C09107=1078.926,391.055,397.098,176.330,30.069,155.273
C09108=1078.920,390.808,397.137,176.326,30.062,155.271
C09109=1078.913,390.562,397.177,176.323,30.054,155.269
C09110=1078.906,390.315,397.216,176.319,30.047,155.268
C09111=1078.900,390.068,397.255,176.314,30.039,155.266
C09112=1078.893,389.821,397.295,176.311,30.032,155.265
C09113=1078.886,389.575,397.333,176.307,30.024,155.263
C09114=1078.880,389.327,397.373,176.303,30.016,155.262
C09115=1078.873,389.081,397.412,176.299,30.009,155.260
C09116=1078.866,388.834,397.451,176.295,30.002,155.259
C09117=1078.860,388.587,397.491,176.291,29.994,155.257
C09118=1078.853,388.340,397.529,176.287,29.986,155.256
C09119=1078.846,388.094,397.569,176.284,29.979,155.254
C09120=1078.840,387.847,397.608,176.279,29.972,155.253
C09121=1078.833,387.600,397.647,176.275,29.964,155.251
C09122=1078.827,387.354,397.686,176.271,29.957,155.250
C09123=1078.821,387.107,397.725,176.268,29.949,155.248
C09124=1078.814,386.860,397.764,176.264,29.942,155.247
C09125=1078.807,386.613,397.803,176.259,29.934,155.245
C09126=1078.801,386.366,397.842,176.256,29.928,155.244
C09127=1078.794,386.119,397.881,176.252,29.920,155.242
C09128=1078.788,385.886,397.918,176.249,29.913,155.241
C09129=1078.782,385.653,397.955,176.245,29.906,155.240
C09130=1078.776,385.419,397.991,176.241,29.899,155.238
C09131=1078.769,385.185,398.029,176.238,29.892,155.237
C09132=1078.764,384.951,398.065,176.234,29.886,155.236
C09133=1078.758,384.718,398.102,176.231,29.879,155.234
C09134=1078.752,384.484,398.139,176.226,29.872,155.233
C09135=1078.746,384.251,398.175,176.223,29.865,155.232
C09136=1078.739,384.004,398.214,176.219,29.858,155.230
C09137=1078.732,383.757,398.252,176.216,29.851,155.229
C09138=1078.726,383.509,398.292,176.211,29.844,155.227
C09139=1078.720,383.263,398.330,176.208,29.837,155.226
C09140=1078.713,383.017,398.369,176.204,29.829,155.224
C09141=1078.707,382.769,398.407,176.200,29.822,155.223
C09142=1078.701,382.523,398.446,176.197,29.815,155.222
C09143=1078.694,382.276,398.485,176.192,29.808,155.220
C09144=1078.688,382.028,398.523,176.189,29.801,155.219
C09145=1078.681,381.782,398.562,176.185,29.794,155.217
C09146=1078.675,381.535,398.601,176.182,29.787,155.216
C09147=1078.668,381.288,398.639,176.178,29.780,155.215
C09148=1078.662,381.041,398.678,176.173,29.773,155.213
C09149=1078.655,380.795,398.715,176.170,29.766,155.212
C09150=1078.648,380.548,398.754,176.166,29.759,155.211
C09151=1078.642,380.300,398.792,176.163,29.752,155.209
C09152=1078.635,380.054,398.830,176.158,29.745,155.208
C09153=1078.629,379.807,398.868,176.155,29.739,155.207
C09154=1078.622,379.559,398.906,176.151,29.731,155.205
C09155=1078.616,379.313,398.945,176.148,29.725,155.204
C09156=1078.610,379.066,398.983,176.144,29.718,155.203
C09157=1078.604,378.819,399.021,176.140,29.711,155.201
C09158=1078.597,378.572,399.060,176.136,29.704,155.200
C09159=1078.591,378.325,399.098,176.133,29.697,155.198
C09160=1078.584,378.078,399.135,176.129,29.691,155.197
C09161=1078.577,377.832,399.174,176.125,29.684,155.196
C09162=1078.571,377.585,399.211,176.121,29.677,155.194
C09163=1078.565,377.337,399.250,176.118,29.670,155.193
C09164=1078.559,377.091,399.287,176.114,29.664,155.192
C09165=1078.552,376.843,399.325,176.111,29.657,155.191
C09166=1078.546,376.596,399.363,176.106,29.650,155.189
C09167=1078.539,376.350,399.401,176.103,29.643,155.188
C09168=1078.533,376.103,399.439,176.099,29.637,155.187
C09169=1078.526,375.856,399.477,176.096,29.630,155.185
C09170=1078.520,375.609,399.515,176.092,29.623,155.184
C09171=1078.514,375.362,399.553,176.088,29.617,155.183
C09172=1078.507,375.115,399.590,176.084,29.610,155.182
C09173=1078.501,374.868,399.628,176.081,29.604,155.180
C09174=1078.495,374.621,399.666,176.077,29.597,155.179
C09175=1078.489,374.374,399.704,176.074,29.590,155.178
C09176=1078.482,374.127,399.742,176.069,29.584,155.176
C09177=1078.476,373.880,399.779,176.066,29.577,155.175
C09178=1078.469,373.633,399.817,176.063,29.571,155.174
C09179=1078.464,373.386,399.854,176.059,29.564,155.173
C09180=1078.456,373.138,399.892,176.055,29.558,155.171
C09181=1078.451,372.892,399.930,176.051,29.551,155.170
C09182=1078.443,372.645,399.967,176.048,29.545,155.169
C09183=1078.437,372.398,400.005,176.044,29.538,155.168
C09184=1078.432,372.178,400.038,176.041,29.533,155.167
C09185=1078.427,371.959,400.071,176.038,29.528,155.166
C09186=1078.420,371.740,400.104,176.035,29.522,155.164
C09187=1078.415,371.520,400.137,176.032,29.516,155.163
C09188=1078.409,371.301,400.171,176.028,29.510,155.162
C09189=1078.404,371.082,400.204,176.025,29.504,155.161
C09190=1078.398,370.862,400.238,176.022,29.499,155.160
C09191=1078.392,370.643,400.269,176.018,29.493,155.159
C09192=1078.386,370.396,400.308,176.015,29.487,155.158
C09193=1078.379,370.149,400.345,176.011,29.481,155.157
C09194=1078.374,369.902,400.382,176.008,29.475,155.156
C09195=1078.366,369.655,400.419,176.004,29.468,155.154
C09196=1078.361,369.407,400.456,176.000,29.462,155.153
C09197=1078.354,369.161,400.493,175.997,29.456,155.152
C09198=1078.348,368.913,400.531,175.993,29.449,155.151
C09199=1078.341,368.666,400.568,175.990,29.443,155.149
C09200=1078.336,368.419,400.605,175.986,29.437,155.148
C09201=1078.329,368.172,400.642,175.982,29.431,155.147
C09202=1078.322,367.925,400.679,175.979,29.424,155.146
C09203=1078.316,367.677,400.716,175.976,29.418,155.145
C09204=1078.310,367.431,400.753,175.972,29.412,155.144
C09205=1078.304,367.184,400.790,175.968,29.406,155.142
C09206=1078.298,366.937,400.827,175.965,29.400,155.141
C09207=1078.292,366.688,400.864,175.961,29.393,155.140
C09208=1078.285,366.442,400.901,175.958,29.387,155.139
C09209=1078.279,366.195,400.938,175.954,29.381,155.138
C09210=1078.273,365.948,400.975,175.950,29.375,155.137
C09211=1078.267,365.701,401.011,175.947,29.369,155.135
C09212=1078.261,365.454,401.049,175.944,29.363,155.134
C09213=1078.254,365.206,401.086,175.940,29.357,155.133
C09214=1078.248,364.959,401.122,175.936,29.351,155.132
C09215=1078.241,364.712,401.159,175.933,29.344,155.131
C09216=1078.236,364.465,401.196,175.930,29.338,155.130
C09217=1078.229,364.218,401.232,175.926,29.333,155.129
C09218=1078.223,363.970,401.269,175.922,29.327,155.128
C09219=1078.216,363.723,401.305,175.919,29.321,155.126
C09220=1078.210,363.476,401.342,175.915,29.314,155.125
C09221=1078.204,363.228,401.379,175.912,29.309,155.124
C09222=1078.198,362.981,401.415,175.908,29.303,155.123
C09223=1078.191,362.734,401.452,175.904,29.296,155.122
C09224=1078.185,362.487,401.488,175.901,29.291,155.121
C09225=1078.179,362.240,401.525,175.898,29.285,155.120
C09226=1078.172,361.993,401.561,175.895,29.279,155.119
C09227=1078.165,361.745,401.598,175.890,29.273,155.118
C09228=1078.160,361.498,401.635,175.887,29.267,155.116
C09229=1078.154,361.250,401.671,175.884,29.261,155.115
C09230=1078.148,361.003,401.707,175.881,29.256,155.114
C09231=1078.141,360.756,401.744,175.876,29.249,155.113
C09232=1078.135,360.509,401.780,175.873,29.244,155.112
C09233=1078.128,360.262,401.817,175.870,29.238,155.111
C09234=1078.122,360.014,401.852,175.867,29.232,155.110
C09235=1078.116,359.767,401.889,175.862,29.226,155.109
C09236=1078.110,359.520,401.925,175.859,29.220,155.108
C09237=1078.104,359.273,401.961,175.856,29.215,155.107
C09238=1078.097,359.026,401.997,175.853,29.209,155.106
C09239=1078.091,358.778,402.034,175.849,29.203,155.105
C09240=1078.086,358.567,402.064,175.846,29.198,155.104
C09241=1078.080,358.356,402.095,175.843,29.193,155.103
C09242=1078.075,358.145,402.126,175.840,29.189,155.102
C09243=1078.070,357.934,402.156,175.837,29.184,155.101
C09244=1078.064,357.722,402.187,175.834,29.178,155.100
C09245=1078.059,357.511,402.218,175.831,29.174,155.099
C09246=1078.053,357.300,402.249,175.828,29.169,155.098
C09247=1078.048,357.089,402.280,175.826,29.164,155.097
C09248=1078.042,356.842,402.315,175.822,29.158,155.096
C09249=1078.036,356.595,402.352,175.818,29.153,155.095
C09250=1078.030,356.347,402.387,175.815,29.147,155.094
C09251=1078.024,356.100,402.424,175.812,29.142,155.093
C09252=1078.018,355.852,402.460,175.809,29.136,155.092
C09253=1078.012,355.604,402.495,175.805,29.131,155.091
C09254=1078.005,355.357,402.532,175.801,29.125,155.090
C09255=1077.998,355.110,402.567,175.798,29.119,155.089
C09256=1077.993,354.863,402.602,175.795,29.114,155.088
C09257=1077.987,354.616,402.639,175.791,29.108,155.087
C09258=1077.981,354.368,402.674,175.788,29.102,155.086
C09259=1077.975,354.121,402.710,175.785,29.097,155.085
C09260=1077.968,353.874,402.747,175.781,29.091,155.084
C09261=1077.962,353.626,402.782,175.777,29.085,155.083
C09262=1077.956,353.379,402.817,175.774,29.080,155.082
C09263=1077.950,353.132,402.853,175.771,29.074,155.081
C09264=1077.944,352.884,402.889,175.768,29.069,155.080
C09265=1077.937,352.637,402.924,175.764,29.063,155.079
C09266=1077.931,352.389,402.960,175.760,29.058,155.078
C09267=1077.925,352.142,402.996,175.757,29.052,155.077
C09268=1077.918,351.894,403.031,175.754,29.047,155.076
C09269=1077.913,351.647,403.066,175.750,29.041,155.075
C09270=1077.907,351.400,403.102,175.747,29.036,155.074
C09271=1077.900,351.152,403.137,175.744,29.031,155.073
C09272=1077.894,350.905,403.173,175.741,29.025,155.072
C09273=1077.888,350.657,403.209,175.737,29.020,155.071
C09274=1077.882,350.410,403.243,175.733,29.014,155.070
C09275=1077.876,350.163,403.279,175.730,29.009,155.069
C09276=1077.869,349.915,403.314,175.727,29.003,155.068
C09277=1077.863,349.668,403.350,175.724,28.998,155.067
C09278=1077.857,349.420,403.384,175.720,28.993,155.066
C09279=1077.851,349.173,403.420,175.717,28.987,155.065
C09280=1077.845,348.925,403.456,175.714,28.982,155.064
C09281=1077.839,348.678,403.490,175.710,28.977,155.064
C09282=1077.833,348.431,403.526,175.707,28.971,155.062
C09283=1077.826,348.183,403.561,175.704,28.966,155.062
C09284=1077.820,347.935,403.596,175.700,28.960,155.061
C09285=1077.814,347.688,403.631,175.697,28.955,155.060
C09286=1077.808,347.441,403.667,175.693,28.950,155.059
C09287=1077.801,347.193,403.702,175.690,28.944,155.058
C09288=1077.796,346.946,403.737,175.687,28.939,155.057
C09289=1077.789,346.698,403.772,175.684,28.934,155.056
C09290=1077.783,346.451,403.807,175.680,28.929,155.055
C09291=1077.778,346.203,403.841,175.677,28.923,155.054
C09292=1077.772,345.956,403.877,175.674,28.918,155.053
C09293=1077.765,345.709,403.912,175.671,28.913,155.052
C09294=1077.759,345.461,403.946,175.667,28.908,155.051
C09295=1077.753,345.213,403.982,175.664,28.903,155.050
C09296=1077.748,345.004,404.011,175.661,28.898,155.050
C09297=1077.743,344.794,404.041,175.658,28.894,155.049
C09298=1077.738,344.585,404.071,175.656,28.889,155.048
C09299=1077.733,344.375,404.100,175.653,28.885,155.047
C09300=1077.727,344.166,404.129,175.650,28.880,155.046
C09301=1077.722,343.956,404.159,175.647,28.876,155.046
C09302=1077.717,343.747,404.188,175.645,28.871,155.045
C09303=1077.712,343.537,404.217,175.641,28.867,155.044
C09304=1077.705,343.290,404.253,175.638,28.862,155.043
C09305=1077.699,343.042,404.287,175.635,28.857,155.042
C09306=1077.693,342.795,404.322,175.631,28.852,155.041
C09307=1077.687,342.547,404.357,175.628,28.847,155.040
C09308=1077.681,342.299,404.391,175.625,28.842,155.040
C09309=1077.674,342.052,404.426,175.622,28.836,155.039
C09310=1077.669,341.804,404.461,175.618,28.831,155.038
C09311=1077.663,341.556,404.495,175.615,28.826,155.037
C09312=1077.656,341.310,404.530,175.612,28.821,155.036
C09313=1077.650,341.062,404.564,175.609,28.816,155.035
C09314=1077.644,340.815,404.598,175.605,28.811,155.034
C09315=1077.638,340.566,404.633,175.602,28.806,155.033
C09316=1077.632,340.320,404.668,175.599,28.801,155.032
C09317=1077.626,340.072,404.702,175.596,28.795,155.031
C09318=1077.620,339.824,404.736,175.592,28.790,155.031
C09319=1077.613,339.576,404.771,175.589,28.786,155.030
C09320=1077.608,339.329,404.806,175.586,28.781,155.029
C09321=1077.602,339.081,404.840,175.582,28.775,155.028
C09322=1077.596,338.833,404.874,175.580,28.771,155.027
C09323=1077.590,338.587,404.909,175.577,28.765,155.026
C09324=1077.583,338.339,404.943,175.574,28.760,155.025
C09325=1077.577,338.092,404.977,175.570,28.756,155.025
C09326=1077.571,337.844,405.012,175.567,28.751,155.024
C09327=1077.565,337.596,405.046,175.564,28.745,155.023
C09328=1077.559,337.348,405.080,175.561,28.741,155.022
C09329=1077.553,337.101,405.114,175.557,28.736,155.021
C09330=1077.547,336.854,405.148,175.554,28.730,155.020
C09331=1077.540,336.606,405.183,175.551,28.726,155.019
C09332=1077.535,336.358,405.216,175.548,28.721,155.018
C09333=1077.528,336.110,405.250,175.544,28.716,155.018
C09334=1077.523,335.863,405.284,175.541,28.711,155.017
C09335=1077.517,335.615,405.319,175.538,28.706,155.016
C09336=1077.510,335.367,405.353,175.535,28.701,155.015
C09337=1077.504,335.120,405.387,175.531,28.696,155.014
C09338=1077.499,334.873,405.421,175.528,28.691,155.013
C09339=1077.492,334.624,405.455,175.525,28.686,155.013
C09340=1077.487,334.377,405.489,175.522,28.682,155.012
C09341=1077.481,334.130,405.523,175.519,28.677,155.011
C09342=1077.474,333.882,405.557,175.516,28.672,155.010
C09343=1077.469,333.634,405.591,175.513,28.667,155.009
C09344=1077.462,333.387,405.624,175.509,28.662,155.008
C09345=1077.456,333.139,405.658,175.506,28.657,155.008
C09346=1077.450,332.891,405.693,175.503,28.652,155.007
C09347=1077.444,332.644,405.726,175.500,28.647,155.006
C09348=1077.438,332.396,405.760,175.496,28.643,155.005
C09349=1077.432,332.148,405.794,175.493,28.637,155.004
C09350=1077.426,331.900,405.828,175.491,28.633,155.003
C09351=1077.420,331.653,405.862,175.488,28.628,155.002
C09352=1077.415,331.441,405.890,175.484,28.624,155.002
C09353=1077.409,331.228,405.919,175.482,28.620,155.001
C09354=1077.404,331.017,405.947,175.479,28.616,155.000
C09355=1077.400,330.804,405.977,175.476,28.612,155.000
C09356=1077.394,330.592,406.005,175.474,28.608,154.999
C09357=1077.388,330.379,406.034,175.471,28.604,154.998
C09358=1077.383,330.167,406.063,175.468,28.599,154.998
C09359=1077.378,329.955,406.091,175.465,28.596,154.997
C09360=1077.372,329.707,406.125,175.462,28.591,154.996
C09361=1077.365,329.460,406.158,175.459,28.586,154.996
C09362=1077.360,329.212,406.192,175.457,28.582,154.995
C09363=1077.353,328.965,406.225,175.453,28.577,154.994
C09364=1077.347,328.716,406.259,175.450,28.573,154.993
C09365=1077.341,328.468,406.292,175.447,28.567,154.992
C09366=1077.335,328.221,406.326,175.443,28.563,154.992
C09367=1077.329,327.974,406.359,175.440,28.558,154.991
C09368=1077.322,327.725,406.392,175.437,28.553,154.990
C09369=1077.316,327.478,406.426,175.435,28.549,154.989
C09370=1077.310,327.230,406.459,175.431,28.544,154.988
C09371=1077.304,326.982,406.492,175.428,28.540,154.988
C09372=1077.298,326.735,406.525,175.425,28.535,154.987
C09373=1077.292,326.488,406.559,175.421,28.530,154.986
C09374=1077.285,326.239,406.592,175.418,28.526,154.985
C09375=1077.280,325.991,406.625,175.416,28.521,154.985
C09376=1077.274,325.744,406.658,175.413,28.517,154.984
C09377=1077.268,325.496,406.692,175.409,28.512,154.983
C09378=1077.261,325.249,406.725,175.406,28.507,154.982
C09379=1077.256,325.001,406.758,175.403,28.503,154.981
C09380=1077.250,324.753,406.791,175.400,28.498,154.981
C09381=1077.243,324.506,406.824,175.397,28.494,154.980
C09382=1077.237,324.257,406.858,175.394,28.489,154.979
C09383=1077.231,324.010,406.890,175.391,28.484,154.978
C09384=1077.225,323.762,406.924,175.387,28.480,154.978
C09385=1077.219,323.514,406.956,175.385,28.475,154.977
C09386=1077.213,323.266,406.990,175.382,28.471,154.976
C09387=1077.207,323.019,407.022,175.379,28.466,154.975
C09388=1077.202,322.771,407.056,175.375,28.461,154.974
C09389=1077.195,322.523,407.089,175.372,28.457,154.974
C09390=1077.189,322.276,407.121,175.370,28.452,154.973
C09391=1077.183,322.028,407.155,175.366,28.447,154.972
C09392=1077.177,321.780,407.187,175.363,28.443,154.971
C09393=1077.172,321.532,407.221,175.360,28.439,154.971
C09394=1077.165,321.285,407.253,175.358,28.434,154.970
C09395=1077.159,321.037,407.286,175.354,28.429,154.969
C09396=1077.154,320.788,407.319,175.351,28.425,154.968
C09397=1077.147,320.541,407.352,175.348,28.420,154.968
C09398=1077.141,320.293,407.384,175.345,28.416,154.967
C09399=1077.136,320.046,407.417,175.342,28.411,154.966
C09400=1077.130,319.798,407.450,175.339,28.406,154.965
C09401=1077.125,319.550,407.483,175.336,28.402,154.965
C09402=1077.118,319.302,407.515,175.333,28.398,154.964
C09403=1077.112,319.055,407.548,175.330,28.393,154.963
C09404=1077.107,318.807,407.581,175.327,28.388,154.962
C09405=1077.101,318.559,407.613,175.324,28.384,154.962
C09406=1077.094,318.311,407.646,175.321,28.379,154.961
C09407=1077.089,318.063,407.680,175.318,28.375,154.960
C09408=1077.084,317.848,407.707,175.316,28.371,154.959
C09409=1077.079,317.633,407.736,175.312,28.367,154.959
C09410=1077.073,317.417,407.764,175.310,28.363,154.958
C09411=1077.068,317.201,407.792,175.307,28.359,154.957
C09412=1077.063,316.986,407.821,175.305,28.355,154.957
C09413=1077.058,316.771,407.849,175.303,28.351,154.956
C09414=1077.054,316.555,407.877,175.299,28.347,154.956
C09415=1077.048,316.340,407.906,175.297,28.343,154.955
C09416=1077.042,316.091,407.938,175.294,28.339,154.954
C09417=1077.037,315.845,407.970,175.291,28.335,154.953
C09418=1077.030,315.597,408.003,175.288,28.330,154.953
C09419=1077.025,315.348,408.036,175.285,28.325,154.952
C09420=1077.019,315.101,408.069,175.283,28.321,154.951
C09421=1077.013,314.853,408.100,175.279,28.317,154.950
C09422=1077.008,314.605,408.133,175.276,28.312,154.950
C09423=1077.001,314.357,408.165,175.273,28.308,154.949
C09424=1076.995,314.109,408.197,175.270,28.303,154.948
C09425=1076.989,313.862,408.230,175.267,28.299,154.948
C09426=1076.983,313.613,408.262,175.264,28.294,154.947
C09427=1076.977,313.366,408.293,175.262,28.291,154.946
C09428=1076.971,313.118,408.326,175.258,28.286,154.946
C09429=1076.965,312.870,408.358,175.255,28.282,154.945
C09430=1076.958,312.622,408.390,175.253,28.278,154.944
C09431=1076.952,312.375,408.422,175.249,28.273,154.943
C09432=1076.946,312.126,408.454,175.246,28.269,154.943
C09433=1076.941,311.879,408.486,175.244,28.265,154.942
C09434=1076.935,311.631,408.518,175.240,28.260,154.941
C09435=1076.928,311.383,408.550,175.237,28.256,154.941
C09436=1076.922,311.135,408.582,175.234,28.251,154.940
C09437=1076.916,310.888,408.614,175.232,28.247,154.939
C09438=1076.910,310.639,408.646,175.228,28.243,154.939
C09439=1076.904,310.392,408.679,175.225,28.239,154.938
C09440=1076.897,310.144,408.710,175.223,28.235,154.937
C09441=1076.892,309.896,408.742,175.219,28.230,154.936
C09442=1076.886,309.648,408.774,175.216,28.226,154.936
C09443=1076.880,309.400,408.806,175.214,28.222,154.935
C09444=1076.875,309.153,408.838,175.210,28.218,154.934
C09445=1076.868,308.905,408.869,175.207,28.213,154.934
C09446=1076.862,308.656,408.901,175.205,28.209,154.933
C09447=1076.856,308.409,408.933,175.202,28.205,154.932
C09448=1076.851,308.161,408.965,175.198,28.200,154.932
C09449=1076.844,307.913,408.996,175.196,28.196,154.931
C09450=1076.838,307.666,409.028,175.193,28.192,154.930
C09451=1076.832,307.418,409.060,175.190,28.187,154.930
C09452=1076.826,307.169,409.091,175.187,28.183,154.929
C09453=1076.820,306.922,409.123,175.184,28.179,154.928
C09454=1076.814,306.673,409.155,175.181,28.175,154.928
C09455=1076.809,306.426,409.187,175.178,28.170,154.927
C09456=1076.802,306.178,409.218,175.175,28.166,154.926
C09457=1076.796,305.930,409.250,175.173,28.162,154.926
C09458=1076.791,305.682,409.282,175.169,28.158,154.925
C09459=1076.784,305.434,409.313,175.166,28.153,154.924
C09460=1076.779,305.187,409.345,175.164,28.149,154.923
C09461=1076.773,304.939,409.377,175.161,28.145,154.923
C09462=1076.767,304.691,409.408,175.158,28.141,154.922
C09463=1076.761,304.443,409.439,175.155,28.136,154.921
C09464=1076.756,304.229,409.466,175.152,28.133,154.921
C09465=1076.751,304.015,409.494,175.150,28.129,154.920
C09466=1076.746,303.802,409.521,175.148,28.126,154.920
C09467=1076.741,303.587,409.548,175.144,28.122,154.919
C09468=1076.736,303.373,409.575,175.142,28.118,154.918
C09469=1076.731,303.160,409.602,175.140,28.115,154.918
C09470=1076.726,302.946,409.630,175.137,28.111,154.917
C09471=1076.721,302.732,409.657,175.135,28.107,154.917
C09472=1076.715,302.484,409.688,175.132,28.103,154.916
C09473=1076.709,302.236,409.719,175.129,28.099,154.915
C09474=1076.702,301.989,409.751,175.126,28.094,154.915
C09475=1076.697,301.740,409.782,175.124,28.090,154.914
C09476=1076.691,301.492,409.814,175.120,28.086,154.913
C09477=1076.686,301.244,409.844,175.118,28.082,154.913
C09478=1076.680,300.997,409.876,175.115,28.078,154.912
C09479=1076.673,300.749,409.907,175.112,28.073,154.911
C09480=1076.668,300.501,409.938,175.109,28.069,154.911
C09481=1076.662,300.253,409.970,175.106,28.065,154.910
C09482=1076.657,300.005,410.001,175.104,28.061,154.909
C09483=1076.651,299.757,410.032,175.100,28.056,154.909
C09484=1076.645,299.509,410.063,175.098,28.053,154.908
C09485=1076.639,299.261,410.095,175.095,28.048,154.907
C09486=1076.634,299.013,410.126,175.092,28.044,154.907
C09487=1076.628,298.765,410.157,175.089,28.040,154.906
C09488=1076.623,298.517,410.188,175.086,28.035,154.905
C09489=1076.616,298.270,410.219,175.084,28.031,154.905
C09490=1076.611,298.021,410.250,175.080,28.027,154.904
C09491=1076.605,297.774,410.281,175.078,28.023,154.903
C09492=1076.599,297.526,410.312,175.075,28.019,154.903
C09493=1076.593,297.277,410.343,175.072,28.015,154.902
C09494=1076.587,297.030,410.374,175.069,28.010,154.901
C09495=1076.581,296.781,410.405,175.066,28.006,154.901
C09496=1076.575,296.533,410.436,175.064,28.002,154.900
C09497=1076.569,296.286,410.467,175.060,27.998,154.899
C09498=1076.564,296.037,410.498,175.058,27.994,154.899
C09499=1076.558,295.789,410.528,175.055,27.990,154.898
C09500=1076.552,295.542,410.559,175.052,27.986,154.897
C09501=1076.545,295.294,410.590,175.049,27.982,154.897
C09502=1076.540,295.046,410.621,175.047,27.978,154.896
C09503=1076.534,294.798,410.652,175.044,27.973,154.895
C09504=1076.528,294.549,410.682,175.041,27.969,154.895
C09505=1076.522,294.301,410.713,175.038,27.965,154.894
C09506=1076.516,294.054,410.744,175.036,27.961,154.893
C09507=1076.510,293.805,410.775,175.032,27.957,154.893
C09508=1076.505,293.558,410.805,175.030,27.953,154.892
C09509=1076.499,293.310,410.836,175.027,27.949,154.892
C09510=1076.493,293.062,410.866,175.024,27.945,154.891
C09511=1076.486,292.813,410.897,175.021,27.941,154.890
C09512=1076.481,292.565,410.928,175.019,27.937,154.890
C09513=1076.476,292.317,410.958,175.016,27.933,154.889
C09514=1076.469,292.069,410.989,175.013,27.929,154.888
C09515=1076.463,291.821,411.019,175.010,27.925,154.888
C09516=1076.458,291.573,411.049,175.008,27.921,154.887
C09517=1076.452,291.325,411.080,175.004,27.916,154.886
C09518=1076.445,291.077,411.111,175.002,27.912,154.886
C09519=1076.439,290.829,411.141,174.999,27.908,154.885
C09520=1076.430,290.416,411.192,174.994,27.902,154.884
C09521=1076.420,290.003,411.242,174.989,27.895,154.883
C09522=1076.411,289.590,411.293,174.985,27.888,154.882
C09523=1076.401,289.176,411.344,174.980,27.881,154.881
C09524=1076.395,288.929,411.374,174.977,27.877,154.880
C09525=1076.389,288.681,411.405,174.975,27.874,154.880
C09526=1076.383,288.432,411.435,174.972,27.870,154.879
C09527=1076.377,288.184,411.465,174.969,27.866,154.879
C09528=1076.371,287.936,411.495,174.967,27.862,154.878
C09529=1076.366,287.688,411.526,174.964,27.857,154.877
C09530=1076.359,287.441,411.555,174.961,27.854,154.877
C09531=1076.353,287.191,411.585,174.958,27.850,154.876
C09532=1076.347,286.944,411.616,174.956,27.846,154.875
C09533=1076.341,286.696,411.646,174.952,27.841,154.875
C09534=1076.336,286.447,411.676,174.950,27.838,154.874
C09535=1076.330,286.200,411.706,174.947,27.834,154.874
C09536=1076.324,285.952,411.736,174.945,27.830,154.873
C09537=1076.319,285.703,411.766,174.941,27.825,154.872
C09538=1076.312,285.455,411.797,174.939,27.822,154.872
C09539=1076.306,285.207,411.827,174.937,27.818,154.871
C09540=1076.300,284.959,411.856,174.933,27.814,154.871
C09541=1076.294,284.711,411.886,174.931,27.810,154.870
C09542=1076.289,284.463,411.916,174.928,27.806,154.869
C09543=1076.283,284.215,411.946,174.925,27.802,154.869
C09544=1076.277,283.967,411.977,174.922,27.798,154.868
C09545=1076.272,283.718,412.006,174.920,27.794,154.867
C09546=1076.265,283.471,412.036,174.917,27.790,154.867
C09547=1076.260,283.222,412.066,174.914,27.786,154.866
C09548=1076.254,282.975,412.096,174.912,27.782,154.866
C09549=1076.248,282.726,412.126,174.909,27.778,154.865
C09550=1076.242,282.478,412.156,174.906,27.774,154.864
C09551=1076.236,282.230,412.185,174.903,27.770,154.864
C09552=1076.231,281.982,412.215,174.901,27.766,154.863
C09553=1076.224,281.733,412.246,174.898,27.762,154.862
C09554=1076.219,281.485,412.275,174.895,27.758,154.862
C09555=1076.214,281.238,412.305,174.893,27.754,154.861
C09556=1076.207,280.990,412.334,174.890,27.750,154.861
C09557=1076.201,280.740,412.364,174.887,27.746,154.860
C09558=1076.195,280.493,412.395,174.885,27.742,154.859
C09559=1076.189,280.245,412.424,174.882,27.738,154.859
C09560=1076.184,279.996,412.453,174.879,27.734,154.858
C09561=1076.178,279.748,412.484,174.876,27.730,154.858
C09562=1076.172,279.500,412.513,174.874,27.727,154.857
C09563=1076.166,279.252,412.542,174.871,27.723,154.856
C09564=1076.161,279.003,412.572,174.868,27.718,154.856
C09565=1076.154,278.756,412.602,174.866,27.715,154.855
C09566=1076.148,278.507,412.631,174.863,27.711,154.855
C09567=1076.142,278.259,412.660,174.860,27.707,154.854
C09568=1076.137,278.011,412.690,174.858,27.703,154.853
C09569=1076.132,277.763,412.719,174.855,27.699,154.853
C09570=1076.125,277.515,412.749,174.852,27.695,154.852
C09571=1076.120,277.267,412.779,174.849,27.691,154.852
C09572=1076.109,276.863,412.826,174.845,27.685,154.851
C09573=1076.100,276.460,412.874,174.841,27.678,154.850
C09574=1076.091,276.057,412.922,174.837,27.672,154.849
C09575=1076.082,275.654,412.970,174.833,27.666,154.848
C09576=1076.076,275.406,412.999,174.829,27.662,154.847
C09577=1076.070,275.157,413.028,174.827,27.658,154.847
C09578=1076.064,274.909,413.057,174.824,27.654,154.846
C09579=1076.058,274.661,413.087,174.822,27.650,154.845
C09580=1076.052,274.412,413.116,174.819,27.646,154.845
C09581=1076.047,274.164,413.146,174.816,27.642,154.844
C09582=1076.041,273.917,413.174,174.814,27.639,154.844
C09583=1076.035,273.668,413.203,174.811,27.634,154.843
C09584=1076.029,273.420,413.233,174.808,27.631,154.842
C09585=1076.023,273.172,413.262,174.806,27.627,154.842
C09586=1076.018,272.923,413.291,174.804,27.623,154.841
C09587=1076.011,272.675,413.320,174.800,27.619,154.841
C09588=1076.005,272.427,413.349,174.798,27.615,154.840
C09589=1076.000,272.178,413.379,174.796,27.611,154.839
C09590=1075.994,271.931,413.407,174.792,27.607,154.839
C09591=1075.988,271.683,413.436,174.790,27.604,154.838
C09592=1075.982,271.434,413.466,174.788,27.600,154.838
C09593=1075.976,271.185,413.494,174.784,27.596,154.837
C09594=1075.970,270.937,413.523,174.782,27.592,154.836
C09595=1075.965,270.689,413.553,174.780,27.588,154.836
C09596=1075.959,270.441,413.582,174.777,27.584,154.835
C09597=1075.953,270.193,413.610,174.774,27.580,154.835
C09598=1075.947,269.944,413.640,174.772,27.577,154.834
C09599=1075.941,269.696,413.669,174.769,27.572,154.833
C09600=1075.936,269.448,413.697,174.766,27.569,154.833
C09601=1075.930,269.200,413.726,174.764,27.565,154.832
C09602=1075.924,268.951,413.755,174.761,27.561,154.832
C09603=1075.918,268.703,413.784,174.759,27.557,154.831
C09604=1075.912,268.455,413.813,174.756,27.554,154.831
C09605=1075.906,268.207,413.841,174.753,27.549,154.830
C09606=1075.900,267.958,413.870,174.751,27.546,154.829
C09607=1075.894,267.710,413.899,174.748,27.542,154.829
C09608=1075.889,267.461,413.928,174.745,27.538,154.828
C09609=1075.883,267.214,413.956,174.743,27.534,154.828
C09610=1075.877,266.966,413.985,174.740,27.530,154.827
C09611=1075.871,266.717,414.014,174.738,27.526,154.826
C09612=1075.865,266.469,414.043,174.735,27.523,154.826
C09613=1075.859,266.221,414.071,174.733,27.519,154.825
C09614=1075.854,265.972,414.100,174.730,27.515,154.825
C09615=1075.848,265.723,414.129,174.727,27.511,154.824
C09616=1075.842,265.476,414.157,174.725,27.507,154.824
C09617=1075.836,265.227,414.186,174.722,27.503,154.823
C09618=1075.830,264.979,414.214,174.720,27.499,154.822
C09619=1075.825,264.731,414.243,174.717,27.496,154.822
C09620=1075.819,264.482,414.271,174.715,27.491,154.821
C09621=1075.813,264.234,414.300,174.712,27.488,154.821
C09622=1075.808,263.986,414.329,174.709,27.484,154.820
C09623=1075.802,263.737,414.357,174.707,27.480,154.820
C09624=1075.792,263.338,414.403,174.703,27.474,154.819
C09625=1075.782,262.937,414.449,174.699,27.468,154.818
C09626=1075.773,262.537,414.494,174.694,27.462,154.817
C09627=1075.763,262.137,414.540,174.690,27.456,154.816
C09628=1075.757,261.889,414.568,174.688,27.452,154.815
C09629=1075.751,261.640,414.596,174.685,27.448,154.815
C09630=1075.746,261.392,414.624,174.682,27.444,154.814
C09631=1075.739,261.144,414.653,174.680,27.441,154.814
C09632=1075.733,260.895,414.681,174.678,27.437,154.813
C09633=1075.728,260.647,414.709,174.674,27.433,154.812
C09634=1075.722,260.398,414.737,174.672,27.430,154.812
C09635=1075.716,260.150,414.766,174.670,27.426,154.811
C09636=1075.709,259.903,414.794,174.668,27.422,154.811
C09637=1075.703,259.654,414.822,174.664,27.418,154.810
C09638=1075.697,259.405,414.850,174.662,27.414,154.810
C09639=1075.692,259.157,414.878,174.660,27.411,154.809
C09640=1075.686,258.908,414.907,174.657,27.407,154.809
C09641=1075.680,258.661,414.934,174.654,27.403,154.808
C09642=1075.674,258.412,414.962,174.652,27.399,154.807
C09643=1075.668,258.163,414.991,174.649,27.396,154.807
C09644=1075.663,257.915,415.019,174.647,27.392,154.806
C09645=1075.656,257.667,415.046,174.644,27.388,154.806
C09646=1075.651,257.418,415.074,174.642,27.384,154.805
C09647=1075.645,257.170,415.103,174.639,27.380,154.805
C09648=1075.639,256.922,415.131,174.637,27.377,154.804
C09649=1075.633,256.673,415.158,174.635,27.373,154.803
C09650=1075.627,256.424,415.187,174.632,27.369,154.803
C09651=1075.622,256.176,415.215,174.629,27.365,154.802
C09652=1075.616,255.928,415.243,174.627,27.362,154.802
C09653=1075.609,255.680,415.270,174.625,27.358,154.801
C09654=1075.604,255.431,415.299,174.621,27.354,154.801
C09655=1075.598,255.183,415.327,174.619,27.350,154.800
C09656=1075.592,254.935,415.354,174.617,27.346,154.799
C09657=1075.586,254.686,415.382,174.615,27.343,154.799
C09658=1075.581,254.437,415.410,174.612,27.339,154.798
C09659=1075.575,254.189,415.438,174.609,27.335,154.798
C09660=1075.569,253.941,415.465,174.607,27.331,154.797
C09661=1075.563,253.693,415.494,174.604,27.327,154.797
C09662=1075.558,253.445,415.522,174.602,27.324,154.796
C09663=1075.551,253.196,415.549,174.600,27.320,154.795
C09664=1075.546,252.948,415.577,174.597,27.316,154.795
C09665=1075.540,252.699,415.605,174.594,27.312,154.794
C09666=1075.534,252.451,415.632,174.592,27.308,154.794
C09667=1075.528,252.202,415.660,174.590,27.304,154.793
C09668=1075.523,251.954,415.688,174.587,27.301,154.793
C09669=1075.517,251.706,415.715,174.584,27.296,154.792
C09670=1075.511,251.457,415.743,174.582,27.293,154.791
C09671=1075.506,251.208,415.771,174.580,27.289,154.791
C09672=1075.500,250.961,415.798,174.577,27.285,154.790
C09673=1075.494,250.711,415.826,174.575,27.282,154.790
C09674=1075.489,250.463,415.854,174.573,27.278,154.789
C09675=1075.482,250.215,415.881,174.570,27.274,154.789
C09676=1075.474,249.812,415.926,174.566,27.268,154.788
C09677=1075.464,249.409,415.971,174.562,27.261,154.787
C09678=1075.455,249.007,416.015,174.558,27.255,154.786
C09679=1075.446,248.604,416.060,174.554,27.249,154.785
C09680=1075.440,248.356,416.087,174.552,27.245,154.784
C09681=1075.435,248.107,416.115,174.549,27.241,154.784
C09682=1075.429,247.859,416.143,174.547,27.238,154.783
C09683=1075.423,247.610,416.170,174.544,27.234,154.782
C09684=1075.418,247.362,416.198,174.542,27.230,154.782
C09685=1075.412,247.114,416.224,174.540,27.226,154.781
C09686=1075.406,246.864,416.252,174.538,27.222,154.781
C09687=1075.400,246.617,416.279,174.535,27.218,154.780
C09688=1075.395,246.368,416.306,174.532,27.215,154.780
C09689=1075.389,246.120,416.334,174.530,27.210,154.779
C09690=1075.383,245.871,416.361,174.527,27.207,154.778
C09691=1075.378,245.623,416.388,174.525,27.203,154.778
C09692=1075.371,245.374,416.416,174.523,27.199,154.777
C09693=1075.366,245.125,416.443,174.521,27.196,154.777
C09694=1075.360,244.877,416.470,174.518,27.192,154.776
C09695=1075.354,244.629,416.497,174.515,27.188,154.776
C09696=1075.349,244.380,416.525,174.513,27.184,154.775
C09697=1075.343,244.132,416.551,174.511,27.180,154.774
C09698=1075.337,243.884,416.579,174.508,27.177,154.774
C09699=1075.332,243.635,416.606,174.506,27.173,154.773
C09700=1075.325,243.386,416.633,174.504,27.169,154.773
C09701=1075.320,243.138,416.660,174.502,27.165,154.772
C09702=1075.314,242.890,416.687,174.498,27.161,154.772
C09703=1075.308,242.641,416.714,174.496,27.157,154.771
C09704=1075.302,242.392,416.741,174.494,27.154,154.770
C09705=1075.297,242.144,416.768,174.492,27.150,154.770
C09706=1075.291,241.895,416.795,174.489,27.146,154.769
C09707=1075.285,241.647,416.822,174.487,27.143,154.769
C09708=1075.279,241.399,416.849,174.485,27.139,154.768
C09709=1075.273,241.150,416.876,174.482,27.135,154.768
C09710=1075.267,240.902,416.903,174.480,27.131,154.767
C09711=1075.262,240.653,416.930,174.477,27.128,154.767
C09712=1075.256,240.404,416.957,174.475,27.123,154.766
C09713=1075.250,240.156,416.984,174.472,27.120,154.765
C09714=1075.244,239.907,417.010,174.470,27.116,154.765
C09715=1075.238,239.659,417.037,174.468,27.112,154.764
C09716=1075.233,239.411,417.064,174.466,27.109,154.764
C09717=1075.226,239.162,417.091,174.463,27.105,154.763
C09718=1075.221,238.913,417.118,174.461,27.101,154.763
C09719=1075.215,238.665,417.144,174.459,27.098,154.762
C09720=1075.210,238.416,417.171,174.456,27.094,154.762
C09721=1075.204,238.168,417.198,174.453,27.090,154.761
C09722=1075.198,237.919,417.224,174.451,27.086,154.760
C09723=1075.192,237.670,417.251,174.449,27.082,154.760
C09724=1075.186,237.422,417.278,174.447,27.079,154.759
C09725=1075.180,237.174,417.305,174.444,27.075,154.759
C09726=1075.174,236.925,417.331,174.442,27.071,154.758
C09727=1075.169,236.677,417.358,174.440,27.067,154.757
C09728=1075.159,236.268,417.401,174.436,27.061,154.757
C09729=1075.150,235.858,417.446,174.432,27.055,154.756
C09730=1075.141,235.449,417.489,174.428,27.049,154.755
C09731=1075.131,235.040,417.533,174.425,27.042,154.754
C09732=1075.125,234.790,417.560,174.422,27.039,154.753
C09733=1075.119,234.542,417.586,174.419,27.035,154.753
C09734=1075.113,234.294,417.613,174.417,27.031,154.752
C09735=1075.107,234.045,417.640,174.415,27.027,154.752
C09736=1075.102,233.796,417.665,174.412,27.023,154.751
C09737=1075.096,233.548,417.692,174.410,27.020,154.750
C09738=1075.090,233.300,417.719,174.408,27.016,154.750
C09739=1075.085,233.051,417.745,174.406,27.012,154.749
C09740=1075.079,232.802,417.771,174.403,27.008,154.749
C09741=1075.073,232.554,417.798,174.401,27.004,154.748
C09742=1075.068,232.306,417.825,174.399,27.001,154.747
C09743=1075.062,232.057,417.851,174.397,26.997,154.747
C09744=1075.056,231.808,417.877,174.394,26.993,154.746
C09745=1075.051,231.559,417.903,174.392,26.990,154.746
C09746=1075.044,231.311,417.929,174.390,26.985,154.745
C09747=1075.039,231.063,417.956,174.388,26.982,154.745
C09748=1075.033,230.814,417.982,174.385,26.978,154.744
C09749=1075.027,230.566,418.008,174.383,26.974,154.743
C09750=1075.022,230.317,418.034,174.381,26.971,154.743
C09751=1075.016,230.068,418.061,174.379,26.967,154.742
C09752=1075.010,229.820,418.086,174.375,26.963,154.742
C09753=1075.004,229.571,418.113,174.373,26.959,154.741
C09754=1074.998,229.323,418.140,174.371,26.955,154.741
C09755=1074.993,229.074,418.166,174.369,26.952,154.740
C09756=1074.986,228.826,418.192,174.366,26.948,154.740
C09757=1074.981,228.577,418.218,174.364,26.944,154.739
C09758=1074.975,228.328,418.244,174.362,26.940,154.738
C09759=1074.969,228.080,418.270,174.360,26.937,154.738
C09760=1074.963,227.831,418.295,174.358,26.933,154.737
C09761=1074.958,227.582,418.322,174.355,26.929,154.737
C09762=1074.951,227.334,418.347,174.353,26.926,154.736
C09763=1074.946,227.085,418.374,174.351,26.921,154.736
C09764=1074.940,226.836,418.400,174.348,26.918,154.735
C09765=1074.934,226.588,418.425,174.346,26.914,154.735
C09766=1074.928,226.339,418.452,174.344,26.910,154.734
C09767=1074.923,226.090,418.478,174.342,26.907,154.733
C09768=1074.917,225.842,418.503,174.340,26.903,154.733
C09769=1074.911,225.593,418.530,174.337,26.899,154.732
C09770=1074.906,225.345,418.556,174.335,26.895,154.732
C09771=1074.900,225.096,418.581,174.333,26.891,154.731
C09772=1074.894,224.848,418.608,174.331,26.888,154.731
C09773=1074.888,224.599,418.633,174.328,26.884,154.730
C09774=1074.882,224.350,418.659,174.326,26.880,154.729
C09775=1074.877,224.101,418.685,174.324,26.877,154.729
C09776=1074.870,223.853,418.711,174.322,26.872,154.728
C09777=1074.865,223.604,418.737,174.319,26.869,154.728
C09778=1074.859,223.356,418.762,174.317,26.865,154.727
C09779=1074.854,223.107,418.788,174.315,26.861,154.727
C09780=1074.844,222.690,418.831,174.311,26.855,154.726
C09781=1074.834,222.272,418.874,174.308,26.849,154.725
C09782=1074.825,221.854,418.918,174.304,26.842,154.724
C09783=1074.815,221.436,418.961,174.300,26.835,154.723
C09784=1074.809,221.188,418.987,174.298,26.832,154.722
C09785=1074.803,220.939,419.013,174.296,26.828,154.722
C09786=1074.798,220.691,419.038,174.293,26.824,154.721
C09787=1074.792,220.442,419.063,174.291,26.821,154.720
C09788=1074.786,220.194,419.089,174.289,26.817,154.720
C09789=1074.780,219.945,419.114,174.287,26.813,154.719
C09790=1074.774,219.696,419.140,174.285,26.809,154.719
C09791=1074.768,219.447,419.165,174.282,26.806,154.718
C09792=1074.762,219.199,419.190,174.280,26.802,154.718
C09793=1074.757,218.950,419.216,174.278,26.798,154.717
C09794=1074.751,218.702,419.242,174.276,26.794,154.717
C09795=1074.744,218.453,419.267,174.273,26.790,154.716
C09796=1074.739,218.204,419.293,174.271,26.787,154.715
C09797=1074.733,217.956,419.318,174.270,26.783,154.715
C09798=1074.728,217.707,419.344,174.268,26.779,154.714
C09799=1074.722,217.459,419.369,174.265,26.776,154.714
C09800=1074.716,217.210,419.395,174.263,26.772,154.713
C09801=1074.711,216.961,419.419,174.261,26.768,154.713
C09802=1074.705,216.712,419.445,174.259,26.764,154.712
C09803=1074.699,216.464,419.470,174.257,26.760,154.711
C09804=1074.693,216.215,419.496,174.254,26.757,154.711
C09805=1074.687,215.967,419.521,174.252,26.753,154.710
C09806=1074.681,215.718,419.546,174.250,26.749,154.710
C09807=1074.675,215.469,419.572,174.248,26.745,154.709
C09808=1074.671,215.220,419.596,174.245,26.741,154.709
C09809=1074.664,214.972,419.622,174.243,26.737,154.708
C09810=1074.658,214.723,419.647,174.241,26.734,154.707
C09811=1074.653,214.475,419.673,174.239,26.730,154.707
C09812=1074.647,214.226,419.697,174.237,26.726,154.706
C09813=1074.641,213.977,419.723,174.234,26.722,154.706
C09814=1074.636,213.729,419.748,174.233,26.719,154.705
C09815=1074.630,213.480,419.774,174.231,26.715,154.705
C09816=1074.624,213.231,419.798,174.229,26.711,154.704
C09817=1074.619,212.983,419.823,174.226,26.707,154.703
C09818=1074.612,212.734,419.849,174.224,26.703,154.703
C09819=1074.607,212.484,419.874,174.222,26.700,154.702
C09820=1074.602,212.236,419.899,174.220,26.695,154.702
C09821=1074.595,211.988,419.924,174.218,26.692,154.701
C09822=1074.589,211.738,419.949,174.216,26.688,154.701
C09823=1074.584,211.490,419.974,174.213,26.684,154.700
C09824=1074.578,211.242,419.999,174.211,26.681,154.699
C09825=1074.572,210.993,420.024,174.209,26.676,154.699
C09826=1074.567,210.744,420.049,174.207,26.673,154.698
C09827=1074.561,210.495,420.074,174.205,26.669,154.698
C09828=1074.555,210.247,420.099,174.203,26.665,154.697
C09829=1074.549,209.998,420.124,174.201,26.661,154.696
C09830=1074.543,209.749,420.149,174.199,26.658,154.696
C09831=1074.538,209.501,420.174,174.197,26.654,154.695
C09832=1074.528,209.088,420.215,174.193,26.648,154.695
C09833=1074.519,208.674,420.256,174.189,26.641,154.693
C09834=1074.509,208.260,420.298,174.186,26.634,154.693
C09835=1074.499,207.847,420.339,174.183,26.628,154.692
C09836=1074.473,206.724,420.447,174.060,26.564,154.691
C09837=1074.469,206.499,420.470,174.058,26.561,154.691
C09838=1074.463,206.274,420.492,174.056,26.559,154.690
C09839=1074.458,206.050,420.514,174.054,26.556,154.690
C09840=1074.451,205.742,420.543,174.052,26.552,154.690
C09841=1074.445,205.434,420.573,174.048,26.549,154.689
C09842=1074.437,205.126,420.603,174.046,26.546,154.689
C09843=1074.430,204.818,420.633,174.043,26.542,154.688
C09844=1074.425,204.569,420.657,174.041,26.539,154.688
C09845=1074.420,204.320,420.680,174.038,26.536,154.688
C09846=1074.413,204.071,420.704,174.036,26.533,154.687
C09847=1074.408,203.823,420.729,174.034,26.531,154.687
C09848=1074.402,203.574,420.753,174.032,26.528,154.686
C09849=1074.396,203.326,420.777,174.030,26.525,154.686
C09850=1074.391,203.076,420.801,174.027,26.522,154.686
C09851=1074.385,202.827,420.825,174.025,26.519,154.685
C09852=1074.379,202.579,420.848,174.023,26.516,154.685
C09853=1074.374,202.330,420.873,174.021,26.514,154.685
C09854=1074.369,202.081,420.897,174.019,26.511,154.684
C09855=1074.363,201.832,420.920,174.016,26.508,154.684
C09856=1074.356,201.584,420.944,174.014,26.505,154.684
C09857=1074.351,201.335,420.968,174.011,26.502,154.683
C09858=1074.345,201.086,420.992,174.009,26.499,154.683
C09859=1074.340,200.837,421.016,174.007,26.497,154.683
C09860=1074.334,200.588,421.039,174.005,26.494,154.682
C09861=1074.329,200.340,421.063,174.003,26.491,154.682
C09862=1074.322,200.091,421.087,174.000,26.488,154.682
C09863=1074.316,199.842,421.110,173.998,26.485,154.681
C09864=1074.311,199.593,421.134,173.996,26.483,154.681
C09865=1074.305,199.345,421.158,173.994,26.480,154.681
C09866=1074.299,199.095,421.182,173.992,26.477,154.680
C09867=1074.293,198.847,421.205,173.989,26.474,154.680
C09868=1074.288,198.598,421.229,173.987,26.472,154.680
C09869=1074.282,198.349,421.253,173.984,26.469,154.679
C09870=1074.276,198.100,421.276,173.983,26.467,154.679
C09871=1074.271,197.851,421.300,173.981,26.463,154.679
C09872=1074.265,197.602,421.323,173.978,26.461,154.678
C09873=1074.259,197.354,421.347,173.976,26.458,154.678
C09874=1074.253,197.105,421.371,173.973,26.455,154.678
C09875=1074.248,196.856,421.394,173.972,26.452,154.677
C09876=1074.243,196.607,421.418,173.970,26.449,154.677
C09877=1074.237,196.359,421.441,173.967,26.447,154.677
C09878=1074.230,196.109,421.465,173.965,26.444,154.676
C09879=1074.225,195.861,421.489,173.962,26.441,154.676
C09880=1074.219,195.612,421.512,173.961,26.438,154.676
C09881=1074.214,195.363,421.536,173.958,26.436,154.675
C09882=1074.208,195.114,421.559,173.956,26.433,154.675
C09883=1074.202,194.866,421.583,173.954,26.430,154.675
C09884=1074.197,194.617,421.606,173.952,26.428,154.674
C09885=1074.192,194.368,421.629,173.950,26.424,154.674
C09886=1074.185,194.119,421.653,173.947,26.422,154.674
C09887=1074.180,193.870,421.677,173.945,26.419,154.673
C09888=1074.174,193.621,421.700,173.943,26.416,154.673
C09889=1074.168,193.373,421.723,173.941,26.413,154.673
C09890=1074.163,193.123,421.747,173.939,26.411,154.672
C09891=1074.157,192.875,421.770,173.937,26.408,154.672
C09892=1074.151,192.626,421.793,173.934,26.405,154.672
C09893=1074.146,192.377,421.817,173.933,26.403,154.671
C09894=1074.141,192.128,421.840,173.930,26.399,154.671
C09895=1074.135,191.880,421.864,173.928,26.397,154.671
C09896=1074.128,191.598,421.890,173.926,26.394,154.670
C09897=1074.123,191.317,421.916,173.923,26.391,154.670
C09898=1074.115,191.036,421.942,173.921,26.388,154.669
C09899=1074.110,190.755,421.968,173.919,26.385,154.669
C09900=1074.105,190.506,421.992,173.916,26.381,154.669
C09901=1074.099,190.257,422.015,173.914,26.378,154.668
C09902=1074.093,190.009,422.039,173.912,26.376,154.668
C09903=1074.087,189.760,422.062,173.910,26.373,154.668
C09904=1074.082,189.511,422.085,173.908,26.370,154.667
C09905=1074.076,189.262,422.108,173.905,26.367,154.667
C09906=1074.071,189.013,422.131,173.904,26.365,154.667
C09907=1074.065,188.764,422.154,173.901,26.362,154.666
C09908=1074.060,188.515,422.178,173.899,26.359,154.666
C09909=1074.054,188.267,422.201,173.897,26.357,154.666
C09910=1074.048,188.018,422.224,173.895,26.354,154.665
C09911=1074.042,187.769,422.247,173.893,26.351,154.665
C09912=1074.037,187.520,422.271,173.890,26.348,154.665
C09913=1074.032,187.271,422.294,173.889,26.345,154.664
C09914=1074.027,187.022,422.316,173.887,26.343,154.664
C09915=1074.021,186.774,422.339,173.884,26.340,154.664
C09916=1074.016,186.524,422.363,173.883,26.337,154.663
C09917=1074.010,186.275,422.386,173.880,26.334,154.663
C09918=1074.004,186.027,422.408,173.878,26.331,154.662
C09919=1073.999,185.778,422.431,173.877,26.329,154.662
C09920=1073.994,185.528,422.455,173.874,26.326,154.662
C09921=1073.988,185.280,422.478,173.872,26.323,154.662
C09922=1073.982,185.031,422.501,173.870,26.320,154.661
C09923=1073.976,184.782,422.524,173.868,26.317,154.661
C09924=1073.971,184.533,422.547,173.866,26.315,154.660
C09925=1073.965,184.284,422.570,173.863,26.312,154.660
C09926=1073.959,184.035,422.593,173.862,26.309,154.660
C09927=1073.953,183.786,422.615,173.859,26.307,154.660
C09928=1073.947,183.538,422.638,173.857,26.304,154.659
C09929=1073.941,183.289,422.661,173.855,26.301,154.659
C09930=1073.936,183.041,422.683,173.853,26.299,154.659
C09931=1073.931,182.791,422.706,173.851,26.296,154.658
C09932=1073.925,182.542,422.729,173.849,26.294,154.658
C09933=1073.919,182.294,422.751,173.847,26.291,154.658
C09934=1073.913,182.045,422.774,173.844,26.288,154.657
C09935=1073.907,181.796,422.797,173.843,26.286,154.657
C09936=1073.901,181.547,422.820,173.840,26.283,154.657
C09937=1073.896,181.297,422.842,173.838,26.281,154.656
C09938=1073.889,181.049,422.864,173.837,26.278,154.656
C09939=1073.884,180.800,422.887,173.834,26.275,154.656
C09940=1073.878,180.551,422.910,173.832,26.272,154.655
C09941=1073.873,180.301,422.933,173.830,26.270,154.655
C09942=1073.866,180.053,422.955,173.828,26.267,154.655
C09943=1073.860,179.804,422.978,173.826,26.264,154.654
C09944=1073.855,179.556,423.000,173.824,26.262,154.654
C09945=1073.850,179.306,423.023,173.822,26.259,154.654
C09946=1073.843,179.058,423.045,173.819,26.256,154.653
C09947=1073.838,178.809,423.068,173.818,26.254,154.653
C09948=1073.832,178.560,423.091,173.815,26.251,154.653
C09949=1073.826,178.310,423.113,173.814,26.249,154.653
C09950=1073.820,178.062,423.135,173.811,26.246,154.652
C09951=1073.814,177.813,423.158,173.809,26.243,154.652
C09952=1073.809,177.564,423.180,173.808,26.241,154.652
C09953=1073.804,177.315,423.203,173.805,26.238,154.651
C09954=1073.798,177.066,423.225,173.803,26.235,154.651
C09955=1073.792,176.817,423.248,173.801,26.233,154.651
C09956=1073.786,176.568,423.271,173.799,26.230,154.650
C09957=1073.781,176.319,423.293,173.797,26.227,154.650
C09958=1073.775,176.071,423.315,173.795,26.224,154.650
C09959=1073.769,175.821,423.337,173.793,26.222,154.649
C09960=1073.762,175.540,423.363,173.790,26.219,154.649
C09961=1073.756,175.258,423.388,173.788,26.216,154.649
C09962=1073.749,174.977,423.413,173.786,26.212,154.648
C09963=1073.744,174.695,423.439,173.783,26.210,154.648
C09964=1073.737,174.447,423.461,173.782,26.207,154.648
C09965=1073.732,174.197,423.483,173.780,26.205,154.647
C09966=1073.727,173.949,423.506,173.778,26.202,154.647
C09967=1073.721,173.700,423.528,173.776,26.199,154.647
C09968=1073.715,173.451,423.550,173.773,26.196,154.646
C09969=1073.709,173.201,423.573,173.772,26.194,154.646
C09970=1073.704,172.953,423.595,173.769,26.191,154.646
C09971=1073.698,172.704,423.617,173.768,26.188,154.645
C09972=1073.693,172.454,423.639,173.766,26.186,154.645
C09973=1073.687,172.207,423.661,173.763,26.183,154.645
C09974=1073.681,171.957,423.683,173.762,26.180,154.644
C09975=1073.676,171.708,423.706,173.760,26.177,154.644
C09976=1073.670,171.459,423.728,173.758,26.175,154.644
C09977=1073.664,171.211,423.751,173.756,26.172,154.643
C09978=1073.659,170.961,423.773,173.754,26.170,154.643
C09979=1073.653,170.712,423.794,173.752,26.167,154.643
C09980=1073.648,170.464,423.817,173.749,26.164,154.642
C09981=1073.642,170.214,423.839,173.748,26.162,154.642
C09982=1073.636,169.965,423.861,173.746,26.159,154.642
C09983=1073.631,169.717,423.883,173.744,26.156,154.641
C09984=1073.626,169.467,423.906,173.742,26.153,154.641
C09985=1073.619,169.218,423.927,173.740,26.151,154.641
C09986=1073.614,168.970,423.950,173.738,26.148,154.640
C09987=1073.608,168.721,423.972,173.736,26.145,154.640
C09988=1073.603,168.472,423.993,173.734,26.143,154.640
C09989=1073.598,168.222,424.016,173.732,26.140,154.639
C09990=1073.591,167.974,424.038,173.730,26.137,154.639
C09991=1073.587,167.725,424.060,173.728,26.135,154.639
C09992=1073.580,167.476,424.081,173.727,26.132,154.638
C09993=1073.575,167.226,424.104,173.724,26.129,154.638
C09994=1073.570,166.978,424.126,173.723,26.126,154.638
C09995=1073.564,166.729,424.148,173.720,26.124,154.637
C09996=1073.559,166.480,424.170,173.718,26.121,154.637
//INST
///DATE 2021/06/25 14:45
///ATTR SC,RW,RJ
////FRAME ROBOT
///GROUP1 RB1
NOP
MOVL C00000 V=800.0 PL=0
MOVL C00001 V=800.0 PL=0
MOVL C00002 V=800.0 PL=0
MOVL C00003 V=800.0 PL=0
MOVL C00004 V=800.0 PL=0
MOVL C00005 V=800.0 PL=0
MOVL C00006 V=800.0 PL=0
MOVL C00007 V=800.0 PL=0
MOVL C00008 V=800.0 PL=0
MOVL C00009 V=800.0 PL=0
MOVL C00010 V=800.0 PL=0
MOVL C00011 V=800.0 PL=0
MOVL C00012 V=800.0 PL=0
MOVL C00013 V=800.0 PL=0
MOVL C00014 V=800.0 PL=0
MOVL C00015 V=800.0 PL=0
MOVL C00016 V=800.0 PL=0
MOVL C00017 V=800.0 PL=0
MOVL C00018 V=800.0 PL=0
MOVL C00019 V=800.0 PL=0
MOVL C00020 V=800.0 PL=0
MOVL C00021 V=800.0 PL=0
MOVL C00022 V=800.0 PL=0
MOVL C00023 V=800.0 PL=0
MOVL C00024 V=800.0 PL=0
MOVL C00025 V=800.0 PL=0
MOVL C00026 V=800.0 PL=0
MOVL C00027 V=800.0 PL=0
MOVL C00028 V=800.0 PL=0
MOVL C00029 V=800.0 PL=0
MOVL C00030 V=800.0 PL=0
MOVL C00031 V=800.0 PL=0
MOVL C00032 V=800.0 PL=0
MOVL C00033 V=800.0 PL=0
MOVL C00034 V=800.0 PL=0
MOVL C00035 V=800.0 PL=0
MOVL C00036 V=800.0 PL=0
MOVL C00037 V=800.0 PL=0
MOVL C00038 V=800.0 PL=0
MOVL C00039 V=800.0 PL=0
MOVL C00040 V=800.0 PL=0
MOVL C00041 V=800.0 PL=0
MOVL C00042 V=800.0 PL=0
MOVL C00043 V=800.0 PL=0
MOVL C00044 V=800.0 PL=0
MOVL C00045 V=800.0 PL=0
MOVL C00046 V=800.0 PL=0
MOVL C00047 V=800.0 PL=0
MOVL C00048 V=800.0 PL=0
MOVL C00049 V=800.0 PL=0
MOVL C00050 V=800.0 PL=0
MOVL C00051 V=800.0 PL=0
MOVL C00052 V=800.0 PL=0
MOVL C00053 V=800.0 PL=0
MOVL C00054 V=800.0 PL=0
MOVL C00055 V=800.0 PL=0
MOVL C00056 V=800.0 PL=0
MOVL C00057 V=800.0 PL=0
MOVL C00058 V=800.0 PL=0
MOVL C00059 V=800.0 PL=0
MOVL C00060 V=800.0 PL=0
MOVL C00061 V=800.0 PL=0
MOVL C00062 V=800.0 PL=0
MOVL C00063 V=800.0 PL=0
MOVL C00064 V=800.0 PL=0
MOVL C00065 V=800.0 PL=0
MOVL C00066 V=800.0 PL=0
MOVL C00067 V=800.0 PL=0
MOVL C00068 V=800.0 PL=0
MOVL C00069 V=800.0 PL=0
MOVL C00070 V=800.0 PL=0
MOVL C00071 V=800.0 PL=0
MOVL C00072 V=800.0 PL=0
MOVL C00073 V=800.0 PL=0
MOVL C00074 V=800.0 PL=0
MOVL C00075 V=800.0 PL=0
MOVL C00076 V=800.0 PL=0
MOVL C00077 V=800.0 PL=0
MOVL C00078 V=800.0 PL=0
MOVL C00079 V=800.0 PL=0
MOVL C00080 V=800.0 PL=0
MOVL C00081 V=800.0 PL=0
MOVL C00082 V=800.0 PL=0
MOVL C00083 V=800.0 PL=0
MOVL C00084 V=800.0 PL=0
MOVL C00085 V=800.0 PL=0
MOVL C00086 V=800.0 PL=0
MOVL C00087 V=800.0 PL=0
MOVL C00088 V=800.0 PL=0
MOVL C00089 V=800.0 PL=0
MOVL C00090 V=800.0 PL=0
MOVL C00091 V=800.0 PL=0
MOVL C00092 V=800.0 PL=0
MOVL C00093 V=800.0 PL=0
MOVL C00094 V=800.0 PL=0
MOVL C00095 V=800.0 PL=0
MOVL C00096 V=800.0 PL=0
MOVL C00097 V=800.0 PL=0
MOVL C00098 V=800.0 PL=0
MOVL C00099 V=800.0 PL=0
MOVL C00100 V=800.0 PL=0
MOVL C00101 V=800.0 PL=0
MOVL C00102 V=800.0 PL=0
MOVL C00103 V=800.0 PL=0
MOVL C00104 V=800.0 PL=0
MOVL C00105 V=800.0 PL=0
MOVL C00106 V=800.0 PL=0
MOVL C00107 V=800.0 PL=0
MOVL C00108 V=800.0 PL=0
MOVL C00109 V=800.0 PL=0
MOVL C00110 V=800.0 PL=0
MOVL C00111 V=800.0 PL=0
MOVL C00112 V=800.0 PL=0
MOVL C00113 V=800.0 PL=0
MOVL C00114 V=800.0 PL=0
MOVL C00115 V=800.0 PL=0
MOVL C00116 V=800.0 PL=0
MOVL C00117 V=800.0 PL=0
MOVL C00118 V=800.0 PL=0
MOVL C00119 V=800.0 PL=0
MOVL C00120 V=800.0 PL=0
MOVL C00121 V=800.0 PL=0
MOVL C00122 V=800.0 PL=0
MOVL C00123 V=800.0 PL=0
MOVL C00124 V=800.0 PL=0
MOVL C00125 V=800.0 PL=0
MOVL C00126 V=800.0 PL=0
MOVL C00127 V=800.0 PL=0
MOVL C00128 V=800.0 PL=0
MOVL C00129 V=800.0 PL=0
MOVL C00130 V=800.0 PL=0
MOVL C00131 V=800.0 PL=0
MOVL C00132 V=800.0 PL=0
MOVL C00133 V=800.0 PL=0
MOVL C00134 V=800.0 PL=0
MOVL C00135 V=800.0 PL=0
MOVL C00136 V=800.0 PL=0
MOVL C00137 V=800.0 PL=0
MOVL C00138 V=800.0 PL=0
MOVL C00139 V=800.0 PL=0
MOVL C00140 V=800.0 PL=0
MOVL C00141 V=800.0 PL=0
MOVL C00142 V=800.0 PL=0
MOVL C00143 V=800.0 PL=0
MOVL C00144 V=800.0 PL=0
MOVL C00145 V=800.0 PL=0
MOVL C00146 V=800.0 PL=0
MOVL C00147 V=800.0 PL=0
MOVL C00148 V=800.0 PL=0
MOVL C00149 V=800.0 PL=0
MOVL C00150 V=800.0 PL=0
MOVL C00151 V=800.0 PL=0
MOVL C00152 V=800.0 PL=0
MOVL C00153 V=800.0 PL=0
MOVL C00154 V=800.0 PL=0
MOVL C00155 V=800.0 PL=0
MOVL C00156 V=800.0 PL=0
MOVL C00157 V=800.0 PL=0
MOVL C00158 V=800.0 PL=0
MOVL C00159 V=800.0 PL=0
MOVL C00160 V=800.0 PL=0
MOVL C00161 V=800.0 PL=0
MOVL C00162 V=800.0 PL=0
MOVL C00163 V=800.0 PL=0
MOVL C00164 V=800.0 PL=0
MOVL C00165 V=800.0 PL=0
MOVL C00166 V=800.0 PL=0
MOVL C00167 V=800.0 PL=0
MOVL C00168 V=800.0 PL=0
MOVL C00169 V=800.0 PL=0
MOVL C00170 V=800.0 PL=0
MOVL C00171 V=800.0 PL=0
MOVL C00172 V=800.0 PL=0
MOVL C00173 V=800.0 PL=0
MOVL C00174 V=800.0 PL=0
MOVL C00175 V=800.0 PL=0
MOVL C00176 V=800.0 PL=0
MOVL C00177 V=800.0 PL=0
MOVL C00178 V=800.0 PL=0
MOVL C00179 V=800.0 PL=0
MOVL C00180 V=800.0 PL=0
MOVL C00181 V=800.0 PL=0
MOVL C00182 V=800.0 PL=0
MOVL C00183 V=800.0 PL=0
MOVL C00184 V=800.0 PL=0
MOVL C00185 V=800.0 PL=0
MOVL C00186 V=800.0 PL=0
MOVL C00187 V=800.0 PL=0
MOVL C00188 V=800.0 PL=0
MOVL C00189 V=800.0 PL=0
MOVL C00190 V=800.0 PL=0
MOVL C00191 V=800.0 PL=0
MOVL C00192 V=800.0 PL=0
MOVL C00193 V=800.0 PL=0
MOVL C00194 V=800.0 PL=0
MOVL C00195 V=800.0 PL=0
MOVL C00196 V=800.0 PL=0
MOVL C00197 V=800.0 PL=0
MOVL C00198 V=800.0 PL=0
MOVL C00199 V=800.0 PL=0
MOVL C00200 V=800.0 PL=0
MOVL C00201 V=800.0 PL=0
MOVL C00202 V=800.0 PL=0
MOVL C00203 V=800.0 PL=0
MOVL C00204 V=800.0 PL=0
MOVL C00205 V=800.0 PL=0
MOVL C00206 V=800.0 PL=0
MOVL C00207 V=800.0 PL=0
MOVL C00208 V=800.0 PL=0
MOVL C00209 V=800.0 PL=0
MOVL C00210 V=800.0 PL=0
MOVL C00211 V=800.0 PL=0
MOVL C00212 V=800.0 PL=0
MOVL C00213 V=800.0 PL=0
MOVL C00214 V=800.0 PL=0
MOVL C00215 V=800.0 PL=0
MOVL C00216 V=800.0 PL=0
MOVL C00217 V=800.0 PL=0
MOVL C00218 V=800.0 PL=0
MOVL C00219 V=800.0 PL=0
MOVL C00220 V=800.0 PL=0
MOVL C00221 V=800.0 PL=0
MOVL C00222 V=800.0 PL=0
MOVL C00223 V=800.0 PL=0
MOVL C00224 V=800.0 PL=0
MOVL C00225 V=800.0 PL=0
MOVL C00226 V=800.0 PL=0
MOVL C00227 V=800.0 PL=0
MOVL C00228 V=800.0 PL=0
MOVL C00229 V=800.0 PL=0
MOVL C00230 V=800.0 PL=0
MOVL C00231 V=800.0 PL=0
MOVL C00232 V=800.0 PL=0
MOVL C00233 V=800.0 PL=0
MOVL C00234 V=800.0 PL=0
MOVL C00235 V=800.0 PL=0
MOVL C00236 V=800.0 PL=0
MOVL C00237 V=800.0 PL=0
MOVL C00238 V=800.0 PL=0
MOVL C00239 V=800.0 PL=0
MOVL C00240 V=800.0 PL=0
MOVL C00241 V=800.0 PL=0
MOVL C00242 V=800.0 PL=0
MOVL C00243 V=800.0 PL=0
MOVL C00244 V=800.0 PL=0
MOVL C00245 V=800.0 PL=0
MOVL C00246 V=800.0 PL=0
MOVL C00247 V=800.0 PL=0
MOVL C00248 V=800.0 PL=0
MOVL C00249 V=800.0 PL=0
MOVL C00250 V=800.0 PL=0
MOVL C00251 V=800.0 PL=0
MOVL C00252 V=800.0 PL=0
MOVL C00253 V=800.0 PL=0
MOVL C00254 V=800.0 PL=0
MOVL C00255 V=800.0 PL=0
MOVL C00256 V=800.0 PL=0
MOVL C00257 V=800.0 PL=0
MOVL C00258 V=800.0 PL=0
MOVL C00259 V=800.0 PL=0
MOVL C00260 V=800.0 PL=0
MOVL C00261 V=800.0 PL=0
MOVL C00262 V=800.0 PL=0
MOVL C00263 V=800.0 PL=0
MOVL C00264 V=800.0 PL=0
MOVL C00265 V=800.0 PL=0
MOVL C00266 V=800.0 PL=0
MOVL C00267 V=800.0 PL=0
MOVL C00268 V=800.0 PL=0
MOVL C00269 V=800.0 PL=0
MOVL C00270 V=800.0 PL=0
MOVL C00271 V=800.0 PL=0
MOVL C00272 V=800.0 PL=0
MOVL C00273 V=800.0 PL=0
MOVL C00274 V=800.0 PL=0
MOVL C00275 V=800.0 PL=0
MOVL C00276 V=800.0 PL=0
MOVL C00277 V=800.0 PL=0
MOVL C00278 V=800.0 PL=0
MOVL C00279 V=800.0 PL=0
MOVL C00280 V=800.0 PL=0
MOVL C00281 V=800.0 PL=0
MOVL C00282 V=800.0 PL=0
MOVL C00283 V=800.0 PL=0
MOVL C00284 V=800.0 PL=0
MOVL C00285 V=800.0 PL=0
MOVL C00286 V=800.0 PL=0
MOVL C00287 V=800.0 PL=0
MOVL C00288 V=800.0 PL=0
MOVL C00289 V=800.0 PL=0
MOVL C00290 V=800.0 PL=0
MOVL C00291 V=800.0 PL=0
MOVL C00292 V=800.0 PL=0
MOVL C00293 V=800.0 PL=0
MOVL C00294 V=800.0 PL=0
MOVL C00295 V=800.0 PL=0
MOVL C00296 V=800.0 PL=0
MOVL C00297 V=800.0 PL=0
MOVL C00298 V=800.0 PL=0
MOVL C00299 V=800.0 PL=0
MOVL C00300 V=800.0 PL=0
MOVL C00301 V=800.0 PL=0
MOVL C00302 V=800.0 PL=0
MOVL C00303 V=800.0 PL=0
MOVL C00304 V=800.0 PL=0
MOVL C00305 V=800.0 PL=0
MOVL C00306 V=800.0 PL=0
MOVL C00307 V=800.0 PL=0
MOVL C00308 V=800.0 PL=0
MOVL C00309 V=800.0 PL=0
MOVL C00310 V=800.0 PL=0
MOVL C00311 V=800.0 PL=0
MOVL C00312 V=800.0 PL=0
MOVL C00313 V=800.0 PL=0
MOVL C00314 V=800.0 PL=0
MOVL C00315 V=800.0 PL=0
MOVL C00316 V=800.0 PL=0
MOVL C00317 V=800.0 PL=0
MOVL C00318 V=800.0 PL=0
MOVL C00319 V=800.0 PL=0
MOVL C00320 V=800.0 PL=0
MOVL C00321 V=800.0 PL=0
MOVL C00322 V=800.0 PL=0
MOVL C00323 V=800.0 PL=0
MOVL C00324 V=800.0 PL=0
MOVL C00325 V=800.0 PL=0
MOVL C00326 V=800.0 PL=0
MOVL C00327 V=800.0 PL=0
MOVL C00328 V=800.0 PL=0
MOVL C00329 V=800.0 PL=0
MOVL C00330 V=800.0 PL=0
MOVL C00331 V=800.0 PL=0
MOVL C00332 V=800.0 PL=0
MOVL C00333 V=800.0 PL=0
MOVL C00334 V=800.0 PL=0
MOVL C00335 V=800.0 PL=0
MOVL C00336 V=800.0 PL=0
MOVL C00337 V=800.0 PL=0
MOVL C00338 V=800.0 PL=0
MOVL C00339 V=800.0 PL=0
MOVL C00340 V=800.0 PL=0
MOVL C00341 V=800.0 PL=0
MOVL C00342 V=800.0 PL=0
MOVL C00343 V=800.0 PL=0
MOVL C00344 V=800.0 PL=0
MOVL C00345 V=800.0 PL=0
MOVL C00346 V=800.0 PL=0
MOVL C00347 V=800.0 PL=0
MOVL C00348 V=800.0 PL=0
MOVL C00349 V=800.0 PL=0
MOVL C00350 V=800.0 PL=0
MOVL C00351 V=800.0 PL=0
MOVL C00352 V=800.0 PL=0
MOVL C00353 V=800.0 PL=0
MOVL C00354 V=800.0 PL=0
MOVL C00355 V=800.0 PL=0
MOVL C00356 V=800.0 PL=0
MOVL C00357 V=800.0 PL=0
MOVL C00358 V=800.0 PL=0
MOVL C00359 V=800.0 PL=0
MOVL C00360 V=800.0 PL=0
MOVL C00361 V=800.0 PL=0
MOVL C00362 V=800.0 PL=0
MOVL C00363 V=800.0 PL=0
MOVL C00364 V=800.0 PL=0
MOVL C00365 V=800.0 PL=0
MOVL C00366 V=800.0 PL=0
MOVL C00367 V=800.0 PL=0
MOVL C00368 V=800.0 PL=0
MOVL C00369 V=800.0 PL=0
MOVL C00370 V=800.0 PL=0
MOVL C00371 V=800.0 PL=0
MOVL C00372 V=800.0 PL=0
MOVL C00373 V=800.0 PL=0
MOVL C00374 V=800.0 PL=0
MOVL C00375 V=800.0 PL=0
MOVL C00376 V=800.0 PL=0
MOVL C00377 V=800.0 PL=0
MOVL C00378 V=800.0 PL=0
MOVL C00379 V=800.0 PL=0
MOVL C00380 V=800.0 PL=0
MOVL C00381 V=800.0 PL=0
MOVL C00382 V=800.0 PL=0
MOVL C00383 V=800.0 PL=0
MOVL C00384 V=800.0 PL=0
MOVL C00385 V=800.0 PL=0
MOVL C00386 V=800.0 PL=0
MOVL C00387 V=800.0 PL=0
MOVL C00388 V=800.0 PL=0
MOVL C00389 V=800.0 PL=0
MOVL C00390 V=800.0 PL=0
MOVL C00391 V=800.0 PL=0
MOVL C00392 V=800.0 PL=0
MOVL C00393 V=800.0 PL=0
MOVL C00394 V=800.0 PL=0
MOVL C00395 V=800.0 PL=0
MOVL C00396 V=800.0 PL=0
MOVL C00397 V=800.0 PL=0
MOVL C00398 V=800.0 PL=0
MOVL C00399 V=800.0 PL=0
MOVL C00400 V=800.0 PL=0
MOVL C00401 V=800.0 PL=0
MOVL C00402 V=800.0 PL=0
MOVL C00403 V=800.0 PL=0
MOVL C00404 V=800.0 PL=0
MOVL C00405 V=800.0 PL=0
MOVL C00406 V=800.0 PL=0
MOVL C00407 V=800.0 PL=0
MOVL C00408 V=800.0 PL=0
MOVL C00409 V=800.0 PL=0
MOVL C00410 V=800.0 PL=0
MOVL C00411 V=800.0 PL=0
MOVL C00412 V=800.0 PL=0
MOVL C00413 V=800.0 PL=0
MOVL C00414 V=800.0 PL=0
MOVL C00415 V=800.0 PL=0
MOVL C00416 V=800.0 PL=0
MOVL C00417 V=800.0 PL=0
MOVL C00418 V=800.0 PL=0
MOVL C00419 V=800.0 PL=0
MOVL C00420 V=800.0 PL=0
MOVL C00421 V=800.0 PL=0
MOVL C00422 V=800.0 PL=0
MOVL C00423 V=800.0 PL=0
MOVL C00424 V=800.0 PL=0
MOVL C00425 V=800.0 PL=0
MOVL C00426 V=800.0 PL=0
MOVL C00427 V=800.0 PL=0
MOVL C00428 V=800.0 PL=0
MOVL C00429 V=800.0 PL=0
MOVL C00430 V=800.0 PL=0
MOVL C00431 V=800.0 PL=0
MOVL C00432 V=800.0 PL=0
MOVL C00433 V=800.0 PL=0
MOVL C00434 V=800.0 PL=0
MOVL C00435 V=800.0 PL=0
MOVL C00436 V=800.0 PL=0
MOVL C00437 V=800.0 PL=0
MOVL C00438 V=800.0 PL=0
MOVL C00439 V=800.0 PL=0
MOVL C00440 V=800.0 PL=0
MOVL C00441 V=800.0 PL=0
MOVL C00442 V=800.0 PL=0
MOVL C00443 V=800.0 PL=0
MOVL C00444 V=800.0 PL=0
MOVL C00445 V=800.0 PL=0
MOVL C00446 V=800.0 PL=0
MOVL C00447 V=800.0 PL=0
MOVL C00448 V=800.0 PL=0
MOVL C00449 V=800.0 PL=0
MOVL C00450 V=800.0 PL=0
MOVL C00451 V=800.0 PL=0
MOVL C00452 V=800.0 PL=0
MOVL C00453 V=800.0 PL=0
MOVL C00454 V=800.0 PL=0
MOVL C00455 V=800.0 PL=0
MOVL C00456 V=800.0 PL=0
MOVL C00457 V=800.0 PL=0
MOVL C00458 V=800.0 PL=0
MOVL C00459 V=800.0 PL=0
MOVL C00460 V=800.0 PL=0
MOVL C00461 V=800.0 PL=0
MOVL C00462 V=800.0 PL=0
MOVL C00463 V=800.0 PL=0
MOVL C00464 V=800.0 PL=0
MOVL C00465 V=800.0 PL=0
MOVL C00466 V=800.0 PL=0
MOVL C00467 V=800.0 PL=0
MOVL C00468 V=800.0 PL=0
MOVL C00469 V=800.0 PL=0
MOVL C00470 V=800.0 PL=0
MOVL C00471 V=800.0 PL=0
MOVL C00472 V=800.0 PL=0
MOVL C00473 V=800.0 PL=0
MOVL C00474 V=800.0 PL=0
MOVL C00475 V=800.0 PL=0
MOVL C00476 V=800.0 PL=0
MOVL C00477 V=800.0 PL=0
MOVL C00478 V=800.0 PL=0
MOVL C00479 V=800.0 PL=0
MOVL C00480 V=800.0 PL=0
MOVL C00481 V=800.0 PL=0
MOVL C00482 V=800.0 PL=0
MOVL C00483 V=800.0 PL=0
MOVL C00484 V=800.0 PL=0
MOVL C00485 V=800.0 PL=0
MOVL C00486 V=800.0 PL=0
MOVL C00487 V=800.0 PL=0
MOVL C00488 V=800.0 PL=0
MOVL C00489 V=800.0 PL=0
MOVL C00490 V=800.0 PL=0
MOVL C00491 V=800.0 PL=0
MOVL C00492 V=800.0 PL=0
MOVL C00493 V=800.0 PL=0
MOVL C00494 V=800.0 PL=0
MOVL C00495 V=800.0 PL=0
MOVL C00496 V=800.0 PL=0
MOVL C00497 V=800.0 PL=0
MOVL C00498 V=800.0 PL=0
MOVL C00499 V=800.0 PL=0
MOVL C00500 V=800.0 PL=0
MOVL C00501 V=800.0 PL=0
MOVL C00502 V=800.0 PL=0
MOVL C00503 V=800.0 PL=0
MOVL C00504 V=800.0 PL=0
MOVL C00505 V=800.0 PL=0
MOVL C00506 V=800.0 PL=0
MOVL C00507 V=800.0 PL=0
MOVL C00508 V=800.0 PL=0
MOVL C00509 V=800.0 PL=0
MOVL C00510 V=800.0 PL=0
MOVL C00511 V=800.0 PL=0
MOVL C00512 V=800.0 PL=0
MOVL C00513 V=800.0 PL=0
MOVL C00514 V=800.0 PL=0
MOVL C00515 V=800.0 PL=0
MOVL C00516 V=800.0 PL=0
MOVL C00517 V=800.0 PL=0
MOVL C00518 V=800.0 PL=0
MOVL C00519 V=800.0 PL=0
MOVL C00520 V=800.0 PL=0
MOVL C00521 V=800.0 PL=0
MOVL C00522 V=800.0 PL=0
MOVL C00523 V=800.0 PL=0
MOVL C00524 V=800.0 PL=0
MOVL C00525 V=800.0 PL=0
MOVL C00526 V=800.0 PL=0
MOVL C00527 V=800.0 PL=0
MOVL C00528 V=800.0 PL=0
MOVL C00529 V=800.0 PL=0
MOVL C00530 V=800.0 PL=0
MOVL C00531 V=800.0 PL=0
MOVL C00532 V=800.0 PL=0
MOVL C00533 V=800.0 PL=0
MOVL C00534 V=800.0 PL=0
MOVL C00535 V=800.0 PL=0
MOVL C00536 V=800.0 PL=0
MOVL C00537 V=800.0 PL=0
MOVL C00538 V=800.0 PL=0
MOVL C00539 V=800.0 PL=0
MOVL C00540 V=800.0 PL=0
MOVL C00541 V=800.0 PL=0
MOVL C00542 V=800.0 PL=0
MOVL C00543 V=800.0 PL=0
MOVL C00544 V=800.0 PL=0
MOVL C00545 V=800.0 PL=0
MOVL C00546 V=800.0 PL=0
MOVL C00547 V=800.0 PL=0
MOVL C00548 V=800.0 PL=0
MOVL C00549 V=800.0 PL=0
MOVL C00550 V=800.0 PL=0
MOVL C00551 V=800.0 PL=0
MOVL C00552 V=800.0 PL=0
MOVL C00553 V=800.0 PL=0
MOVL C00554 V=800.0 PL=0
MOVL C00555 V=800.0 PL=0
MOVL C00556 V=800.0 PL=0
MOVL C00557 V=800.0 PL=0
MOVL C00558 V=800.0 PL=0
MOVL C00559 V=800.0 PL=0
MOVL C00560 V=800.0 PL=0
MOVL C00561 V=800.0 PL=0
MOVL C00562 V=800.0 PL=0
MOVL C00563 V=800.0 PL=0
MOVL C00564 V=800.0 PL=0
MOVL C00565 V=800.0 PL=0
MOVL C00566 V=800.0 PL=0
MOVL C00567 V=800.0 PL=0
MOVL C00568 V=800.0 PL=0
MOVL C00569 V=800.0 PL=0
MOVL C00570 V=800.0 PL=0
MOVL C00571 V=800.0 PL=0
MOVL C00572 V=800.0 PL=0
MOVL C00573 V=800.0 PL=0
MOVL C00574 V=800.0 PL=0
MOVL C00575 V=800.0 PL=0
MOVL C00576 V=800.0 PL=0
MOVL C00577 V=800.0 PL=0
MOVL C00578 V=800.0 PL=0
MOVL C00579 V=800.0 PL=0
MOVL C00580 V=800.0 PL=0
MOVL C00581 V=800.0 PL=0
MOVL C00582 V=800.0 PL=0
MOVL C00583 V=800.0 PL=0
MOVL C00584 V=800.0 PL=0
MOVL C00585 V=800.0 PL=0
MOVL C00586 V=800.0 PL=0
MOVL C00587 V=800.0 PL=0
MOVL C00588 V=800.0 PL=0
MOVL C00589 V=800.0 PL=0
MOVL C00590 V=800.0 PL=0
MOVL C00591 V=800.0 PL=0
MOVL C00592 V=800.0 PL=0
MOVL C00593 V=800.0 PL=0
MOVL C00594 V=800.0 PL=0
MOVL C00595 V=800.0 PL=0
MOVL C00596 V=800.0 PL=0
MOVL C00597 V=800.0 PL=0
MOVL C00598 V=800.0 PL=0
MOVL C00599 V=800.0 PL=0
MOVL C00600 V=800.0 PL=0
MOVL C00601 V=800.0 PL=0
MOVL C00602 V=800.0 PL=0
MOVL C00603 V=800.0 PL=0
MOVL C00604 V=800.0 PL=0
MOVL C00605 V=800.0 PL=0
MOVL C00606 V=800.0 PL=0
MOVL C00607 V=800.0 PL=0
MOVL C00608 V=800.0 PL=0
MOVL C00609 V=800.0 PL=0
MOVL C00610 V=800.0 PL=0
MOVL C00611 V=800.0 PL=0
MOVL C00612 V=800.0 PL=0
MOVL C00613 V=800.0 PL=0
MOVL C00614 V=800.0 PL=0
MOVL C00615 V=800.0 PL=0
MOVL C00616 V=800.0 PL=0
MOVL C00617 V=800.0 PL=0
MOVL C00618 V=800.0 PL=0
MOVL C00619 V=800.0 PL=0
MOVL C00620 V=800.0 PL=0
MOVL C00621 V=800.0 PL=0
MOVL C00622 V=800.0 PL=0
MOVL C00623 V=800.0 PL=0
MOVL C00624 V=800.0 PL=0
MOVL C00625 V=800.0 PL=0
MOVL C00626 V=800.0 PL=0
MOVL C00627 V=800.0 PL=0
MOVL C00628 V=800.0 PL=0
MOVL C00629 V=800.0 PL=0
MOVL C00630 V=800.0 PL=0
MOVL C00631 V=800.0 PL=0
MOVL C00632 V=800.0 PL=0
MOVL C00633 V=800.0 PL=0
MOVL C00634 V=800.0 PL=0
MOVL C00635 V=800.0 PL=0
MOVL C00636 V=800.0 PL=0
MOVL C00637 V=800.0 PL=0
MOVL C00638 V=800.0 PL=0
MOVL C00639 V=800.0 PL=0
MOVL C00640 V=800.0 PL=0
MOVL C00641 V=800.0 PL=0
MOVL C00642 V=800.0 PL=0
MOVL C00643 V=800.0 PL=0
MOVL C00644 V=800.0 PL=0
MOVL C00645 V=800.0 PL=0
MOVL C00646 V=800.0 PL=0
MOVL C00647 V=800.0 PL=0
MOVL C00648 V=800.0 PL=0
MOVL C00649 V=800.0 PL=0
MOVL C00650 V=800.0 PL=0
MOVL C00651 V=800.0 PL=0
MOVL C00652 V=800.0 PL=0
MOVL C00653 V=800.0 PL=0
MOVL C00654 V=800.0 PL=0
MOVL C00655 V=800.0 PL=0
MOVL C00656 V=800.0 PL=0
MOVL C00657 V=800.0 PL=0
MOVL C00658 V=800.0 PL=0
MOVL C00659 V=800.0 PL=0
MOVL C00660 V=800.0 PL=0
MOVL C00661 V=800.0 PL=0
MOVL C00662 V=800.0 PL=0
MOVL C00663 V=800.0 PL=0
MOVL C00664 V=800.0 PL=0
MOVL C00665 V=800.0 PL=0
MOVL C00666 V=800.0 PL=0
MOVL C00667 V=800.0 PL=0
MOVL C00668 V=800.0 PL=0
MOVL C00669 V=800.0 PL=0
MOVL C00670 V=800.0 PL=0
MOVL C00671 V=800.0 PL=0
MOVL C00672 V=800.0 PL=0
MOVL C00673 V=800.0 PL=0
MOVL C00674 V=800.0 PL=0
MOVL C00675 V=800.0 PL=0
MOVL C00676 V=800.0 PL=0
MOVL C00677 V=800.0 PL=0
MOVL C00678 V=800.0 PL=0
MOVL C00679 V=800.0 PL=0
MOVL C00680 V=800.0 PL=0
MOVL C00681 V=800.0 PL=0
MOVL C00682 V=800.0 PL=0
MOVL C00683 V=800.0 PL=0
MOVL C00684 V=800.0 PL=0
MOVL C00685 V=800.0 PL=0
MOVL C00686 V=800.0 PL=0
MOVL C00687 V=800.0 PL=0
MOVL C00688 V=800.0 PL=0
MOVL C00689 V=800.0 PL=0
MOVL C00690 V=800.0 PL=0
MOVL C00691 V=800.0 PL=0
MOVL C00692 V=800.0 PL=0
MOVL C00693 V=800.0 PL=0
MOVL C00694 V=800.0 PL=0
MOVL C00695 V=800.0 PL=0
MOVL C00696 V=800.0 PL=0
MOVL C00697 V=800.0 PL=0
MOVL C00698 V=800.0 PL=0
MOVL C00699 V=800.0 PL=0
MOVL C00700 V=800.0 PL=0
MOVL C00701 V=800.0 PL=0
MOVL C00702 V=800.0 PL=0
MOVL C00703 V=800.0 PL=0
MOVL C00704 V=800.0 PL=0
MOVL C00705 V=800.0 PL=0
MOVL C00706 V=800.0 PL=0
MOVL C00707 V=800.0 PL=0
MOVL C00708 V=800.0 PL=0
MOVL C00709 V=800.0 PL=0
MOVL C00710 V=800.0 PL=0
MOVL C00711 V=800.0 PL=0
MOVL C00712 V=800.0 PL=0
MOVL C00713 V=800.0 PL=0
MOVL C00714 V=800.0 PL=0
MOVL C00715 V=800.0 PL=0
MOVL C00716 V=800.0 PL=0
MOVL C00717 V=800.0 PL=0
MOVL C00718 V=800.0 PL=0
MOVL C00719 V=800.0 PL=0
MOVL C00720 V=800.0 PL=0
MOVL C00721 V=800.0 PL=0
MOVL C00722 V=800.0 PL=0
MOVL C00723 V=800.0 PL=0
MOVL C00724 V=800.0 PL=0
MOVL C00725 V=800.0 PL=0
MOVL C00726 V=800.0 PL=0
MOVL C00727 V=800.0 PL=0
MOVL C00728 V=800.0 PL=0
MOVL C00729 V=800.0 PL=0
MOVL C00730 V=800.0 PL=0
MOVL C00731 V=800.0 PL=0
MOVL C00732 V=800.0 PL=0
MOVL C00733 V=800.0 PL=0
MOVL C00734 V=800.0 PL=0
MOVL C00735 V=800.0 PL=0
MOVL C00736 V=800.0 PL=0
MOVL C00737 V=800.0 PL=0
MOVL C00738 V=800.0 PL=0
MOVL C00739 V=800.0 PL=0
MOVL C00740 V=800.0 PL=0
MOVL C00741 V=800.0 PL=0
MOVL C00742 V=800.0 PL=0
MOVL C00743 V=800.0 PL=0
MOVL C00744 V=800.0 PL=0
MOVL C00745 V=800.0 PL=0
MOVL C00746 V=800.0 PL=0
MOVL C00747 V=800.0 PL=0
MOVL C00748 V=800.0 PL=0
MOVL C00749 V=800.0 PL=0
MOVL C00750 V=800.0 PL=0
MOVL C00751 V=800.0 PL=0
MOVL C00752 V=800.0 PL=0
MOVL C00753 V=800.0 PL=0
MOVL C00754 V=800.0 PL=0
MOVL C00755 V=800.0 PL=0
MOVL C00756 V=800.0 PL=0
MOVL C00757 V=800.0 PL=0
MOVL C00758 V=800.0 PL=0
MOVL C00759 V=800.0 PL=0
MOVL C00760 V=800.0 PL=0
MOVL C00761 V=800.0 PL=0
MOVL C00762 V=800.0 PL=0
MOVL C00763 V=800.0 PL=0
MOVL C00764 V=800.0 PL=0
MOVL C00765 V=800.0 PL=0
MOVL C00766 V=800.0 PL=0
MOVL C00767 V=800.0 PL=0
MOVL C00768 V=800.0 PL=0
MOVL C00769 V=800.0 PL=0
MOVL C00770 V=800.0 PL=0
MOVL C00771 V=800.0 PL=0
MOVL C00772 V=800.0 PL=0
MOVL C00773 V=800.0 PL=0
MOVL C00774 V=800.0 PL=0
MOVL C00775 V=800.0 PL=0
MOVL C00776 V=800.0 PL=0
MOVL C00777 V=800.0 PL=0
MOVL C00778 V=800.0 PL=0
MOVL C00779 V=800.0 PL=0
MOVL C00780 V=800.0 PL=0
MOVL C00781 V=800.0 PL=0
MOVL C00782 V=800.0 PL=0
MOVL C00783 V=800.0 PL=0
MOVL C00784 V=800.0 PL=0
MOVL C00785 V=800.0 PL=0
MOVL C00786 V=800.0 PL=0
MOVL C00787 V=800.0 PL=0
MOVL C00788 V=800.0 PL=0
MOVL C00789 V=800.0 PL=0
MOVL C00790 V=800.0 PL=0
MOVL C00791 V=800.0 PL=0
MOVL C00792 V=800.0 PL=0
MOVL C00793 V=800.0 PL=0
MOVL C00794 V=800.0 PL=0
MOVL C00795 V=800.0 PL=0
MOVL C00796 V=800.0 PL=0
MOVL C00797 V=800.0 PL=0
MOVL C00798 V=800.0 PL=0
MOVL C00799 V=800.0 PL=0
MOVL C00800 V=800.0 PL=0
MOVL C00801 V=800.0 PL=0
MOVL C00802 V=800.0 PL=0
MOVL C00803 V=800.0 PL=0
MOVL C00804 V=800.0 PL=0
MOVL C00805 V=800.0 PL=0
MOVL C00806 V=800.0 PL=0
MOVL C00807 V=800.0 PL=0
MOVL C00808 V=800.0 PL=0
MOVL C00809 V=800.0 PL=0
MOVL C00810 V=800.0 PL=0
MOVL C00811 V=800.0 PL=0
MOVL C00812 V=800.0 PL=0
MOVL C00813 V=800.0 PL=0
MOVL C00814 V=800.0 PL=0
MOVL C00815 V=800.0 PL=0
MOVL C00816 V=800.0 PL=0
MOVL C00817 V=800.0 PL=0
MOVL C00818 V=800.0 PL=0
MOVL C00819 V=800.0 PL=0
MOVL C00820 V=800.0 PL=0
MOVL C00821 V=800.0 PL=0
MOVL C00822 V=800.0 PL=0
MOVL C00823 V=800.0 PL=0
MOVL C00824 V=800.0 PL=0
MOVL C00825 V=800.0 PL=0
MOVL C00826 V=800.0 PL=0
MOVL C00827 V=800.0 PL=0
MOVL C00828 V=800.0 PL=0
MOVL C00829 V=800.0 PL=0
MOVL C00830 V=800.0 PL=0
MOVL C00831 V=800.0 PL=0
MOVL C00832 V=800.0 PL=0
MOVL C00833 V=800.0 PL=0
MOVL C00834 V=800.0 PL=0
MOVL C00835 V=800.0 PL=0
MOVL C00836 V=800.0 PL=0
MOVL C00837 V=800.0 PL=0
MOVL C00838 V=800.0 PL=0
MOVL C00839 V=800.0 PL=0
MOVL C00840 V=800.0 PL=0
MOVL C00841 V=800.0 PL=0
MOVL C00842 V=800.0 PL=0
MOVL C00843 V=800.0 PL=0
MOVL C00844 V=800.0 PL=0
MOVL C00845 V=800.0 PL=0
MOVL C00846 V=800.0 PL=0
MOVL C00847 V=800.0 PL=0
MOVL C00848 V=800.0 PL=0
MOVL C00849 V=800.0 PL=0
MOVL C00850 V=800.0 PL=0
MOVL C00851 V=800.0 PL=0
MOVL C00852 V=800.0 PL=0
MOVL C00853 V=800.0 PL=0
MOVL C00854 V=800.0 PL=0
MOVL C00855 V=800.0 PL=0
MOVL C00856 V=800.0 PL=0
MOVL C00857 V=800.0 PL=0
MOVL C00858 V=800.0 PL=0
MOVL C00859 V=800.0 PL=0
MOVL C00860 V=800.0 PL=0
MOVL C00861 V=800.0 PL=0
MOVL C00862 V=800.0 PL=0
MOVL C00863 V=800.0 PL=0
MOVL C00864 V=800.0 PL=0
MOVL C00865 V=800.0 PL=0
MOVL C00866 V=800.0 PL=0
MOVL C00867 V=800.0 PL=0
MOVL C00868 V=800.0 PL=0
MOVL C00869 V=800.0 PL=0
MOVL C00870 V=800.0 PL=0
MOVL C00871 V=800.0 PL=0
MOVL C00872 V=800.0 PL=0
MOVL C00873 V=800.0 PL=0
MOVL C00874 V=800.0 PL=0
MOVL C00875 V=800.0 PL=0
MOVL C00876 V=800.0 PL=0
MOVL C00877 V=800.0 PL=0
MOVL C00878 V=800.0 PL=0
MOVL C00879 V=800.0 PL=0
MOVL C00880 V=800.0 PL=0
MOVL C00881 V=800.0 PL=0
MOVL C00882 V=800.0 PL=0
MOVL C00883 V=800.0 PL=0
MOVL C00884 V=800.0 PL=0
MOVL C00885 V=800.0 PL=0
MOVL C00886 V=800.0 PL=0
MOVL C00887 V=800.0 PL=0
MOVL C00888 V=800.0 PL=0
MOVL C00889 V=800.0 PL=0
MOVL C00890 V=800.0 PL=0
MOVL C00891 V=800.0 PL=0
MOVL C00892 V=800.0 PL=0
MOVL C00893 V=800.0 PL=0
MOVL C00894 V=800.0 PL=0
MOVL C00895 V=800.0 PL=0
MOVL C00896 V=800.0 PL=0
MOVL C00897 V=800.0 PL=0
MOVL C00898 V=800.0 PL=0
MOVL C00899 V=800.0 PL=0
MOVL C00900 V=800.0 PL=0
MOVL C00901 V=800.0 PL=0
MOVL C00902 V=800.0 PL=0
MOVL C00903 V=800.0 PL=0
MOVL C00904 V=800.0 PL=0
MOVL C00905 V=800.0 PL=0
MOVL C00906 V=800.0 PL=0
MOVL C00907 V=800.0 PL=0
MOVL C00908 V=800.0 PL=0
MOVL C00909 V=800.0 PL=0
MOVL C00910 V=800.0 PL=0
MOVL C00911 V=800.0 PL=0
MOVL C00912 V=800.0 PL=0
MOVL C00913 V=800.0 PL=0
MOVL C00914 V=800.0 PL=0
MOVL C00915 V=800.0 PL=0
MOVL C00916 V=800.0 PL=0
MOVL C00917 V=800.0 PL=0
MOVL C00918 V=800.0 PL=0
MOVL C00919 V=800.0 PL=0
MOVL C00920 V=800.0 PL=0
MOVL C00921 V=800.0 PL=0
MOVL C00922 V=800.0 PL=0
MOVL C00923 V=800.0 PL=0
MOVL C00924 V=800.0 PL=0
MOVL C00925 V=800.0 PL=0
MOVL C00926 V=800.0 PL=0
MOVL C00927 V=800.0 PL=0
MOVL C00928 V=800.0 PL=0
MOVL C00929 V=800.0 PL=0
MOVL C00930 V=800.0 PL=0
MOVL C00931 V=800.0 PL=0
MOVL C00932 V=800.0 PL=0
MOVL C00933 V=800.0 PL=0
MOVL C00934 V=800.0 PL=0
MOVL C00935 V=800.0 PL=0
MOVL C00936 V=800.0 PL=0
MOVL C00937 V=800.0 PL=0
MOVL C00938 V=800.0 PL=0
MOVL C00939 V=800.0 PL=0
MOVL C00940 V=800.0 PL=0
MOVL C00941 V=800.0 PL=0
MOVL C00942 V=800.0 PL=0
MOVL C00943 V=800.0 PL=0
MOVL C00944 V=800.0 PL=0
MOVL C00945 V=800.0 PL=0
MOVL C00946 V=800.0 PL=0
MOVL C00947 V=800.0 PL=0
MOVL C00948 V=800.0 PL=0
MOVL C00949 V=800.0 PL=0
MOVL C00950 V=800.0 PL=0
MOVL C00951 V=800.0 PL=0
MOVL C00952 V=800.0 PL=0
MOVL C00953 V=800.0 PL=0
MOVL C00954 V=800.0 PL=0
MOVL C00955 V=800.0 PL=0
MOVL C00956 V=800.0 PL=0
MOVL C00957 V=800.0 PL=0
MOVL C00958 V=800.0 PL=0
MOVL C00959 V=800.0 PL=0
MOVL C00960 V=800.0 PL=0
MOVL C00961 V=800.0 PL=0
MOVL C00962 V=800.0 PL=0
MOVL C00963 V=800.0 PL=0
MOVL C00964 V=800.0 PL=0
MOVL C00965 V=800.0 PL=0
MOVL C00966 V=800.0 PL=0
MOVL C00967 V=800.0 PL=0
MOVL C00968 V=800.0 PL=0
MOVL C00969 V=800.0 PL=0
MOVL C00970 V=800.0 PL=0
MOVL C00971 V=800.0 PL=0
MOVL C00972 V=800.0 PL=0
MOVL C00973 V=800.0 PL=0
MOVL C00974 V=800.0 PL=0
MOVL C00975 V=800.0 PL=0
MOVL C00976 V=800.0 PL=0
MOVL C00977 V=800.0 PL=0
MOVL C00978 V=800.0 PL=0
MOVL C00979 V=800.0 PL=0
MOVL C00980 V=800.0 PL=0
MOVL C00981 V=800.0 PL=0
MOVL C00982 V=800.0 PL=0
MOVL C00983 V=800.0 PL=0
MOVL C00984 V=800.0 PL=0
MOVL C00985 V=800.0 PL=0
MOVL C00986 V=800.0 PL=0
MOVL C00987 V=800.0 PL=0
MOVL C00988 V=800.0 PL=0
MOVL C00989 V=800.0 PL=0
MOVL C00990 V=800.0 PL=0
MOVL C00991 V=800.0 PL=0
MOVL C00992 V=800.0 PL=0
MOVL C00993 V=800.0 PL=0
MOVL C00994 V=800.0 PL=0
MOVL C00995 V=800.0 PL=0
MOVL C00996 V=800.0 PL=0
MOVL C00997 V=800.0 PL=0
MOVL C00998 V=800.0 PL=0
MOVL C00999 V=800.0 PL=0
MOVL C01000 V=800.0 PL=0
MOVL C01001 V=800.0 PL=0
MOVL C01002 V=800.0 PL=0
MOVL C01003 V=800.0 PL=0
MOVL C01004 V=800.0 PL=0
MOVL C01005 V=800.0 PL=0
MOVL C01006 V=800.0 PL=0
MOVL C01007 V=800.0 PL=0
MOVL C01008 V=800.0 PL=0
MOVL C01009 V=800.0 PL=0
MOVL C01010 V=800.0 PL=0
MOVL C01011 V=800.0 PL=0
MOVL C01012 V=800.0 PL=0
MOVL C01013 V=800.0 PL=0
MOVL C01014 V=800.0 PL=0
MOVL C01015 V=800.0 PL=0
MOVL C01016 V=800.0 PL=0
MOVL C01017 V=800.0 PL=0
MOVL C01018 V=800.0 PL=0
MOVL C01019 V=800.0 PL=0
MOVL C01020 V=800.0 PL=0
MOVL C01021 V=800.0 PL=0
MOVL C01022 V=800.0 PL=0
MOVL C01023 V=800.0 PL=0
MOVL C01024 V=800.0 PL=0
MOVL C01025 V=800.0 PL=0
MOVL C01026 V=800.0 PL=0
MOVL C01027 V=800.0 PL=0
MOVL C01028 V=800.0 PL=0
MOVL C01029 V=800.0 PL=0
MOVL C01030 V=800.0 PL=0
MOVL C01031 V=800.0 PL=0
MOVL C01032 V=800.0 PL=0
MOVL C01033 V=800.0 PL=0
MOVL C01034 V=800.0 PL=0
MOVL C01035 V=800.0 PL=0
MOVL C01036 V=800.0 PL=0
MOVL C01037 V=800.0 PL=0
MOVL C01038 V=800.0 PL=0
MOVL C01039 V=800.0 PL=0
MOVL C01040 V=800.0 PL=0
MOVL C01041 V=800.0 PL=0
MOVL C01042 V=800.0 PL=0
MOVL C01043 V=800.0 PL=0
MOVL C01044 V=800.0 PL=0
MOVL C01045 V=800.0 PL=0
MOVL C01046 V=800.0 PL=0
MOVL C01047 V=800.0 PL=0
MOVL C01048 V=800.0 PL=0
MOVL C01049 V=800.0 PL=0
MOVL C01050 V=800.0 PL=0
MOVL C01051 V=800.0 PL=0
MOVL C01052 V=800.0 PL=0
MOVL C01053 V=800.0 PL=0
MOVL C01054 V=800.0 PL=0
MOVL C01055 V=800.0 PL=0
MOVL C01056 V=800.0 PL=0
MOVL C01057 V=800.0 PL=0
MOVL C01058 V=800.0 PL=0
MOVL C01059 V=800.0 PL=0
MOVL C01060 V=800.0 PL=0
MOVL C01061 V=800.0 PL=0
MOVL C01062 V=800.0 PL=0
MOVL C01063 V=800.0 PL=0
MOVL C01064 V=800.0 PL=0
MOVL C01065 V=800.0 PL=0
MOVL C01066 V=800.0 PL=0
MOVL C01067 V=800.0 PL=0
MOVL C01068 V=800.0 PL=0
MOVL C01069 V=800.0 PL=0
MOVL C01070 V=800.0 PL=0
MOVL C01071 V=800.0 PL=0
MOVL C01072 V=800.0 PL=0
MOVL C01073 V=800.0 PL=0
MOVL C01074 V=800.0 PL=0
MOVL C01075 V=800.0 PL=0
MOVL C01076 V=800.0 PL=0
MOVL C01077 V=800.0 PL=0
MOVL C01078 V=800.0 PL=0
MOVL C01079 V=800.0 PL=0
MOVL C01080 V=800.0 PL=0
MOVL C01081 V=800.0 PL=0
MOVL C01082 V=800.0 PL=0
MOVL C01083 V=800.0 PL=0
MOVL C01084 V=800.0 PL=0
MOVL C01085 V=800.0 PL=0
MOVL C01086 V=800.0 PL=0
MOVL C01087 V=800.0 PL=0
MOVL C01088 V=800.0 PL=0
MOVL C01089 V=800.0 PL=0
MOVL C01090 V=800.0 PL=0
MOVL C01091 V=800.0 PL=0
MOVL C01092 V=800.0 PL=0
MOVL C01093 V=800.0 PL=0
MOVL C01094 V=800.0 PL=0
MOVL C01095 V=800.0 PL=0
MOVL C01096 V=800.0 PL=0
MOVL C01097 V=800.0 PL=0
MOVL C01098 V=800.0 PL=0
MOVL C01099 V=800.0 PL=0
MOVL C01100 V=800.0 PL=0
MOVL C01101 V=800.0 PL=0
MOVL C01102 V=800.0 PL=0
MOVL C01103 V=800.0 PL=0
MOVL C01104 V=800.0 PL=0
MOVL C01105 V=800.0 PL=0
MOVL C01106 V=800.0 PL=0
MOVL C01107 V=800.0 PL=0
MOVL C01108 V=800.0 PL=0
MOVL C01109 V=800.0 PL=0
MOVL C01110 V=800.0 PL=0
MOVL C01111 V=800.0 PL=0
MOVL C01112 V=800.0 PL=0
MOVL C01113 V=800.0 PL=0
MOVL C01114 V=800.0 PL=0
MOVL C01115 V=800.0 PL=0
MOVL C01116 V=800.0 PL=0
MOVL C01117 V=800.0 PL=0
MOVL C01118 V=800.0 PL=0
MOVL C01119 V=800.0 PL=0
MOVL C01120 V=800.0 PL=0
MOVL C01121 V=800.0 PL=0
MOVL C01122 V=800.0 PL=0
MOVL C01123 V=800.0 PL=0
MOVL C01124 V=800.0 PL=0
MOVL C01125 V=800.0 PL=0
MOVL C01126 V=800.0 PL=0
MOVL C01127 V=800.0 PL=0
MOVL C01128 V=800.0 PL=0
MOVL C01129 V=800.0 PL=0
MOVL C01130 V=800.0 PL=0
MOVL C01131 V=800.0 PL=0
MOVL C01132 V=800.0 PL=0
MOVL C01133 V=800.0 PL=0
MOVL C01134 V=800.0 PL=0
MOVL C01135 V=800.0 PL=0
MOVL C01136 V=800.0 PL=0
MOVL C01137 V=800.0 PL=0
MOVL C01138 V=800.0 PL=0
MOVL C01139 V=800.0 PL=0
MOVL C01140 V=800.0 PL=0
MOVL C01141 V=800.0 PL=0
MOVL C01142 V=800.0 PL=0
MOVL C01143 V=800.0 PL=0
MOVL C01144 V=800.0 PL=0
MOVL C01145 V=800.0 PL=0
MOVL C01146 V=800.0 PL=0
MOVL C01147 V=800.0 PL=0
MOVL C01148 V=800.0 PL=0
MOVL C01149 V=800.0 PL=0
MOVL C01150 V=800.0 PL=0
MOVL C01151 V=800.0 PL=0
MOVL C01152 V=800.0 PL=0
MOVL C01153 V=800.0 PL=0
MOVL C01154 V=800.0 PL=0
MOVL C01155 V=800.0 PL=0
MOVL C01156 V=800.0 PL=0
MOVL C01157 V=800.0 PL=0
MOVL C01158 V=800.0 PL=0
MOVL C01159 V=800.0 PL=0
MOVL C01160 V=800.0 PL=0
MOVL C01161 V=800.0 PL=0
MOVL C01162 V=800.0 PL=0
MOVL C01163 V=800.0 PL=0
MOVL C01164 V=800.0 PL=0
MOVL C01165 V=800.0 PL=0
MOVL C01166 V=800.0 PL=0
MOVL C01167 V=800.0 PL=0
MOVL C01168 V=800.0 PL=0
MOVL C01169 V=800.0 PL=0
MOVL C01170 V=800.0 PL=0
MOVL C01171 V=800.0 PL=0
MOVL C01172 V=800.0 PL=0
MOVL C01173 V=800.0 PL=0
MOVL C01174 V=800.0 PL=0
MOVL C01175 V=800.0 PL=0
MOVL C01176 V=800.0 PL=0
MOVL C01177 V=800.0 PL=0
MOVL C01178 V=800.0 PL=0
MOVL C01179 V=800.0 PL=0
MOVL C01180 V=800.0 PL=0
MOVL C01181 V=800.0 PL=0
MOVL C01182 V=800.0 PL=0
MOVL C01183 V=800.0 PL=0
MOVL C01184 V=800.0 PL=0
MOVL C01185 V=800.0 PL=0
MOVL C01186 V=800.0 PL=0
MOVL C01187 V=800.0 PL=0
MOVL C01188 V=800.0 PL=0
MOVL C01189 V=800.0 PL=0
MOVL C01190 V=800.0 PL=0
MOVL C01191 V=800.0 PL=0
MOVL C01192 V=800.0 PL=0
MOVL C01193 V=800.0 PL=0
MOVL C01194 V=800.0 PL=0
MOVL C01195 V=800.0 PL=0
MOVL C01196 V=800.0 PL=0
MOVL C01197 V=800.0 PL=0
MOVL C01198 V=800.0 PL=0
MOVL C01199 V=800.0 PL=0
MOVL C01200 V=800.0 PL=0
MOVL C01201 V=800.0 PL=0
MOVL C01202 V=800.0 PL=0
MOVL C01203 V=800.0 PL=0
MOVL C01204 V=800.0 PL=0
MOVL C01205 V=800.0 PL=0
MOVL C01206 V=800.0 PL=0
MOVL C01207 V=800.0 PL=0
MOVL C01208 V=800.0 PL=0
MOVL C01209 V=800.0 PL=0
MOVL C01210 V=800.0 PL=0
MOVL C01211 V=800.0 PL=0
MOVL C01212 V=800.0 PL=0
MOVL C01213 V=800.0 PL=0
MOVL C01214 V=800.0 PL=0
MOVL C01215 V=800.0 PL=0
MOVL C01216 V=800.0 PL=0
MOVL C01217 V=800.0 PL=0
MOVL C01218 V=800.0 PL=0
MOVL C01219 V=800.0 PL=0
MOVL C01220 V=800.0 PL=0
MOVL C01221 V=800.0 PL=0
MOVL C01222 V=800.0 PL=0
MOVL C01223 V=800.0 PL=0
MOVL C01224 V=800.0 PL=0
MOVL C01225 V=800.0 PL=0
MOVL C01226 V=800.0 PL=0
MOVL C01227 V=800.0 PL=0
MOVL C01228 V=800.0 PL=0
MOVL C01229 V=800.0 PL=0
MOVL C01230 V=800.0 PL=0
MOVL C01231 V=800.0 PL=0
MOVL C01232 V=800.0 PL=0
MOVL C01233 V=800.0 PL=0
MOVL C01234 V=800.0 PL=0
MOVL C01235 V=800.0 PL=0
MOVL C01236 V=800.0 PL=0
MOVL C01237 V=800.0 PL=0
MOVL C01238 V=800.0 PL=0
MOVL C01239 V=800.0 PL=0
MOVL C01240 V=800.0 PL=0
MOVL C01241 V=800.0 PL=0
MOVL C01242 V=800.0 PL=0
MOVL C01243 V=800.0 PL=0
MOVL C01244 V=800.0 PL=0
MOVL C01245 V=800.0 PL=0
MOVL C01246 V=800.0 PL=0
MOVL C01247 V=800.0 PL=0
MOVL C01248 V=800.0 PL=0
MOVL C01249 V=800.0 PL=0
MOVL C01250 V=800.0 PL=0
MOVL C01251 V=800.0 PL=0
MOVL C01252 V=800.0 PL=0
MOVL C01253 V=800.0 PL=0
MOVL C01254 V=800.0 PL=0
MOVL C01255 V=800.0 PL=0
MOVL C01256 V=800.0 PL=0
MOVL C01257 V=800.0 PL=0
MOVL C01258 V=800.0 PL=0
MOVL C01259 V=800.0 PL=0
MOVL C01260 V=800.0 PL=0
MOVL C01261 V=800.0 PL=0
MOVL C01262 V=800.0 PL=0
MOVL C01263 V=800.0 PL=0
MOVL C01264 V=800.0 PL=0
MOVL C01265 V=800.0 PL=0
MOVL C01266 V=800.0 PL=0
MOVL C01267 V=800.0 PL=0
MOVL C01268 V=800.0 PL=0
MOVL C01269 V=800.0 PL=0
MOVL C01270 V=800.0 PL=0
MOVL C01271 V=800.0 PL=0
MOVL C01272 V=800.0 PL=0
MOVL C01273 V=800.0 PL=0
MOVL C01274 V=800.0 PL=0
MOVL C01275 V=800.0 PL=0
MOVL C01276 V=800.0 PL=0
MOVL C01277 V=800.0 PL=0
MOVL C01278 V=800.0 PL=0
MOVL C01279 V=800.0 PL=0
MOVL C01280 V=800.0 PL=0
MOVL C01281 V=800.0 PL=0
MOVL C01282 V=800.0 PL=0
MOVL C01283 V=800.0 PL=0
MOVL C01284 V=800.0 PL=0
MOVL C01285 V=800.0 PL=0
MOVL C01286 V=800.0 PL=0
MOVL C01287 V=800.0 PL=0
MOVL C01288 V=800.0 PL=0
MOVL C01289 V=800.0 PL=0
MOVL C01290 V=800.0 PL=0
MOVL C01291 V=800.0 PL=0
MOVL C01292 V=800.0 PL=0
MOVL C01293 V=800.0 PL=0
MOVL C01294 V=800.0 PL=0
MOVL C01295 V=800.0 PL=0
MOVL C01296 V=800.0 PL=0
MOVL C01297 V=800.0 PL=0
MOVL C01298 V=800.0 PL=0
MOVL C01299 V=800.0 PL=0
MOVL C01300 V=800.0 PL=0
MOVL C01301 V=800.0 PL=0
MOVL C01302 V=800.0 PL=0
MOVL C01303 V=800.0 PL=0
MOVL C01304 V=800.0 PL=0
MOVL C01305 V=800.0 PL=0
MOVL C01306 V=800.0 PL=0
MOVL C01307 V=800.0 PL=0
MOVL C01308 V=800.0 PL=0
MOVL C01309 V=800.0 PL=0
MOVL C01310 V=800.0 PL=0
MOVL C01311 V=800.0 PL=0
MOVL C01312 V=800.0 PL=0
MOVL C01313 V=800.0 PL=0
MOVL C01314 V=800.0 PL=0
MOVL C01315 V=800.0 PL=0
MOVL C01316 V=800.0 PL=0
MOVL C01317 V=800.0 PL=0
MOVL C01318 V=800.0 PL=0
MOVL C01319 V=800.0 PL=0
MOVL C01320 V=800.0 PL=0
MOVL C01321 V=800.0 PL=0
MOVL C01322 V=800.0 PL=0
MOVL C01323 V=800.0 PL=0
MOVL C01324 V=800.0 PL=0
MOVL C01325 V=800.0 PL=0
MOVL C01326 V=800.0 PL=0
MOVL C01327 V=800.0 PL=0
MOVL C01328 V=800.0 PL=0
MOVL C01329 V=800.0 PL=0
MOVL C01330 V=800.0 PL=0
MOVL C01331 V=800.0 PL=0
MOVL C01332 V=800.0 PL=0
MOVL C01333 V=800.0 PL=0
MOVL C01334 V=800.0 PL=0
MOVL C01335 V=800.0 PL=0
MOVL C01336 V=800.0 PL=0
MOVL C01337 V=800.0 PL=0
MOVL C01338 V=800.0 PL=0
MOVL C01339 V=800.0 PL=0
MOVL C01340 V=800.0 PL=0
MOVL C01341 V=800.0 PL=0
MOVL C01342 V=800.0 PL=0
MOVL C01343 V=800.0 PL=0
MOVL C01344 V=800.0 PL=0
MOVL C01345 V=800.0 PL=0
MOVL C01346 V=800.0 PL=0
MOVL C01347 V=800.0 PL=0
MOVL C01348 V=800.0 PL=0
MOVL C01349 V=800.0 PL=0
MOVL C01350 V=800.0 PL=0
MOVL C01351 V=800.0 PL=0
MOVL C01352 V=800.0 PL=0
MOVL C01353 V=800.0 PL=0
MOVL C01354 V=800.0 PL=0
MOVL C01355 V=800.0 PL=0
MOVL C01356 V=800.0 PL=0
MOVL C01357 V=800.0 PL=0
MOVL C01358 V=800.0 PL=0
MOVL C01359 V=800.0 PL=0
MOVL C01360 V=800.0 PL=0
MOVL C01361 V=800.0 PL=0
MOVL C01362 V=800.0 PL=0
MOVL C01363 V=800.0 PL=0
MOVL C01364 V=800.0 PL=0
MOVL C01365 V=800.0 PL=0
MOVL C01366 V=800.0 PL=0
MOVL C01367 V=800.0 PL=0
MOVL C01368 V=800.0 PL=0
MOVL C01369 V=800.0 PL=0
MOVL C01370 V=800.0 PL=0
MOVL C01371 V=800.0 PL=0
MOVL C01372 V=800.0 PL=0
MOVL C01373 V=800.0 PL=0
MOVL C01374 V=800.0 PL=0
MOVL C01375 V=800.0 PL=0
MOVL C01376 V=800.0 PL=0
MOVL C01377 V=800.0 PL=0
MOVL C01378 V=800.0 PL=0
MOVL C01379 V=800.0 PL=0
MOVL C01380 V=800.0 PL=0
MOVL C01381 V=800.0 PL=0
MOVL C01382 V=800.0 PL=0
MOVL C01383 V=800.0 PL=0
MOVL C01384 V=800.0 PL=0
MOVL C01385 V=800.0 PL=0
MOVL C01386 V=800.0 PL=0
MOVL C01387 V=800.0 PL=0
MOVL C01388 V=800.0 PL=0
MOVL C01389 V=800.0 PL=0
MOVL C01390 V=800.0 PL=0
MOVL C01391 V=800.0 PL=0
MOVL C01392 V=800.0 PL=0
MOVL C01393 V=800.0 PL=0
MOVL C01394 V=800.0 PL=0
MOVL C01395 V=800.0 PL=0
MOVL C01396 V=800.0 PL=0
MOVL C01397 V=800.0 PL=0
MOVL C01398 V=800.0 PL=0
MOVL C01399 V=800.0 PL=0
MOVL C01400 V=800.0 PL=0
MOVL C01401 V=800.0 PL=0
MOVL C01402 V=800.0 PL=0
MOVL C01403 V=800.0 PL=0
MOVL C01404 V=800.0 PL=0
MOVL C01405 V=800.0 PL=0
MOVL C01406 V=800.0 PL=0
MOVL C01407 V=800.0 PL=0
MOVL C01408 V=800.0 PL=0
MOVL C01409 V=800.0 PL=0
MOVL C01410 V=800.0 PL=0
MOVL C01411 V=800.0 PL=0
MOVL C01412 V=800.0 PL=0
MOVL C01413 V=800.0 PL=0
MOVL C01414 V=800.0 PL=0
MOVL C01415 V=800.0 PL=0
MOVL C01416 V=800.0 PL=0
MOVL C01417 V=800.0 PL=0
MOVL C01418 V=800.0 PL=0
MOVL C01419 V=800.0 PL=0
MOVL C01420 V=800.0 PL=0
MOVL C01421 V=800.0 PL=0
MOVL C01422 V=800.0 PL=0
MOVL C01423 V=800.0 PL=0
MOVL C01424 V=800.0 PL=0
MOVL C01425 V=800.0 PL=0
MOVL C01426 V=800.0 PL=0
MOVL C01427 V=800.0 PL=0
MOVL C01428 V=800.0 PL=0
MOVL C01429 V=800.0 PL=0
MOVL C01430 V=800.0 PL=0
MOVL C01431 V=800.0 PL=0
MOVL C01432 V=800.0 PL=0
MOVL C01433 V=800.0 PL=0
MOVL C01434 V=800.0 PL=0
MOVL C01435 V=800.0 PL=0
MOVL C01436 V=800.0 PL=0
MOVL C01437 V=800.0 PL=0
MOVL C01438 V=800.0 PL=0
MOVL C01439 V=800.0 PL=0
MOVL C01440 V=800.0 PL=0
MOVL C01441 V=800.0 PL=0
MOVL C01442 V=800.0 PL=0
MOVL C01443 V=800.0 PL=0
MOVL C01444 V=800.0 PL=0
MOVL C01445 V=800.0 PL=0
MOVL C01446 V=800.0 PL=0
MOVL C01447 V=800.0 PL=0
MOVL C01448 V=800.0 PL=0
MOVL C01449 V=800.0 PL=0
MOVL C01450 V=800.0 PL=0
MOVL C01451 V=800.0 PL=0
MOVL C01452 V=800.0 PL=0
MOVL C01453 V=800.0 PL=0
MOVL C01454 V=800.0 PL=0
MOVL C01455 V=800.0 PL=0
MOVL C01456 V=800.0 PL=0
MOVL C01457 V=800.0 PL=0
MOVL C01458 V=800.0 PL=0
MOVL C01459 V=800.0 PL=0
MOVL C01460 V=800.0 PL=0
MOVL C01461 V=800.0 PL=0
MOVL C01462 V=800.0 PL=0
MOVL C01463 V=800.0 PL=0
MOVL C01464 V=800.0 PL=0
MOVL C01465 V=800.0 PL=0
MOVL C01466 V=800.0 PL=0
MOVL C01467 V=800.0 PL=0
MOVL C01468 V=800.0 PL=0
MOVL C01469 V=800.0 PL=0
MOVL C01470 V=800.0 PL=0
MOVL C01471 V=800.0 PL=0
MOVL C01472 V=800.0 PL=0
MOVL C01473 V=800.0 PL=0
MOVL C01474 V=800.0 PL=0
MOVL C01475 V=800.0 PL=0
MOVL C01476 V=800.0 PL=0
MOVL C01477 V=800.0 PL=0
MOVL C01478 V=800.0 PL=0
MOVL C01479 V=800.0 PL=0
MOVL C01480 V=800.0 PL=0
MOVL C01481 V=800.0 PL=0
MOVL C01482 V=800.0 PL=0
MOVL C01483 V=800.0 PL=0
MOVL C01484 V=800.0 PL=0
MOVL C01485 V=800.0 PL=0
MOVL C01486 V=800.0 PL=0
MOVL C01487 V=800.0 PL=0
MOVL C01488 V=800.0 PL=0
MOVL C01489 V=800.0 PL=0
MOVL C01490 V=800.0 PL=0
MOVL C01491 V=800.0 PL=0
MOVL C01492 V=800.0 PL=0
MOVL C01493 V=800.0 PL=0
MOVL C01494 V=800.0 PL=0
MOVL C01495 V=800.0 PL=0
MOVL C01496 V=800.0 PL=0
MOVL C01497 V=800.0 PL=0
MOVL C01498 V=800.0 PL=0
MOVL C01499 V=800.0 PL=0
MOVL C01500 V=800.0 PL=0
MOVL C01501 V=800.0 PL=0
MOVL C01502 V=800.0 PL=0
MOVL C01503 V=800.0 PL=0
MOVL C01504 V=800.0 PL=0
MOVL C01505 V=800.0 PL=0
MOVL C01506 V=800.0 PL=0
MOVL C01507 V=800.0 PL=0
MOVL C01508 V=800.0 PL=0
MOVL C01509 V=800.0 PL=0
MOVL C01510 V=800.0 PL=0
MOVL C01511 V=800.0 PL=0
MOVL C01512 V=800.0 PL=0
MOVL C01513 V=800.0 PL=0
MOVL C01514 V=800.0 PL=0
MOVL C01515 V=800.0 PL=0
MOVL C01516 V=800.0 PL=0
MOVL C01517 V=800.0 PL=0
MOVL C01518 V=800.0 PL=0
MOVL C01519 V=800.0 PL=0
MOVL C01520 V=800.0 PL=0
MOVL C01521 V=800.0 PL=0
MOVL C01522 V=800.0 PL=0
MOVL C01523 V=800.0 PL=0
MOVL C01524 V=800.0 PL=0
MOVL C01525 V=800.0 PL=0
MOVL C01526 V=800.0 PL=0
MOVL C01527 V=800.0 PL=0
MOVL C01528 V=800.0 PL=0
MOVL C01529 V=800.0 PL=0
MOVL C01530 V=800.0 PL=0
MOVL C01531 V=800.0 PL=0
MOVL C01532 V=800.0 PL=0
MOVL C01533 V=800.0 PL=0
MOVL C01534 V=800.0 PL=0
MOVL C01535 V=800.0 PL=0
MOVL C01536 V=800.0 PL=0
MOVL C01537 V=800.0 PL=0
MOVL C01538 V=800.0 PL=0
MOVL C01539 V=800.0 PL=0
MOVL C01540 V=800.0 PL=0
MOVL C01541 V=800.0 PL=0
MOVL C01542 V=800.0 PL=0
MOVL C01543 V=800.0 PL=0
MOVL C01544 V=800.0 PL=0
MOVL C01545 V=800.0 PL=0
MOVL C01546 V=800.0 PL=0
MOVL C01547 V=800.0 PL=0
MOVL C01548 V=800.0 PL=0
MOVL C01549 V=800.0 PL=0
MOVL C01550 V=800.0 PL=0
MOVL C01551 V=800.0 PL=0
MOVL C01552 V=800.0 PL=0
MOVL C01553 V=800.0 PL=0
MOVL C01554 V=800.0 PL=0
MOVL C01555 V=800.0 PL=0
MOVL C01556 V=800.0 PL=0
MOVL C01557 V=800.0 PL=0
MOVL C01558 V=800.0 PL=0
MOVL C01559 V=800.0 PL=0
MOVL C01560 V=800.0 PL=0
MOVL C01561 V=800.0 PL=0
MOVL C01562 V=800.0 PL=0
MOVL C01563 V=800.0 PL=0
MOVL C01564 V=800.0 PL=0
MOVL C01565 V=800.0 PL=0
MOVL C01566 V=800.0 PL=0
MOVL C01567 V=800.0 PL=0
MOVL C01568 V=800.0 PL=0
MOVL C01569 V=800.0 PL=0
MOVL C01570 V=800.0 PL=0
MOVL C01571 V=800.0 PL=0
MOVL C01572 V=800.0 PL=0
MOVL C01573 V=800.0 PL=0
MOVL C01574 V=800.0 PL=0
MOVL C01575 V=800.0 PL=0
MOVL C01576 V=800.0 PL=0
MOVL C01577 V=800.0 PL=0
MOVL C01578 V=800.0 PL=0
MOVL C01579 V=800.0 PL=0
MOVL C01580 V=800.0 PL=0
MOVL C01581 V=800.0 PL=0
MOVL C01582 V=800.0 PL=0
MOVL C01583 V=800.0 PL=0
MOVL C01584 V=800.0 PL=0
MOVL C01585 V=800.0 PL=0
MOVL C01586 V=800.0 PL=0
MOVL C01587 V=800.0 PL=0
MOVL C01588 V=800.0 PL=0
MOVL C01589 V=800.0 PL=0
MOVL C01590 V=800.0 PL=0
MOVL C01591 V=800.0 PL=0
MOVL C01592 V=800.0 PL=0
MOVL C01593 V=800.0 PL=0
MOVL C01594 V=800.0 PL=0
MOVL C01595 V=800.0 PL=0
MOVL C01596 V=800.0 PL=0
MOVL C01597 V=800.0 PL=0
MOVL C01598 V=800.0 PL=0
MOVL C01599 V=800.0 PL=0
MOVL C01600 V=800.0 PL=0
MOVL C01601 V=800.0 PL=0
MOVL C01602 V=800.0 PL=0
MOVL C01603 V=800.0 PL=0
MOVL C01604 V=800.0 PL=0
MOVL C01605 V=800.0 PL=0
MOVL C01606 V=800.0 PL=0
MOVL C01607 V=800.0 PL=0
MOVL C01608 V=800.0 PL=0
MOVL C01609 V=800.0 PL=0
MOVL C01610 V=800.0 PL=0
MOVL C01611 V=800.0 PL=0
MOVL C01612 V=800.0 PL=0
MOVL C01613 V=800.0 PL=0
MOVL C01614 V=800.0 PL=0
MOVL C01615 V=800.0 PL=0
MOVL C01616 V=800.0 PL=0
MOVL C01617 V=800.0 PL=0
MOVL C01618 V=800.0 PL=0
MOVL C01619 V=800.0 PL=0
MOVL C01620 V=800.0 PL=0
MOVL C01621 V=800.0 PL=0
MOVL C01622 V=800.0 PL=0
MOVL C01623 V=800.0 PL=0
MOVL C01624 V=800.0 PL=0
MOVL C01625 V=800.0 PL=0
MOVL C01626 V=800.0 PL=0
MOVL C01627 V=800.0 PL=0
MOVL C01628 V=800.0 PL=0
MOVL C01629 V=800.0 PL=0
MOVL C01630 V=800.0 PL=0
MOVL C01631 V=800.0 PL=0
MOVL C01632 V=800.0 PL=0
MOVL C01633 V=800.0 PL=0
MOVL C01634 V=800.0 PL=0
MOVL C01635 V=800.0 PL=0
MOVL C01636 V=800.0 PL=0
MOVL C01637 V=800.0 PL=0
MOVL C01638 V=800.0 PL=0
MOVL C01639 V=800.0 PL=0
MOVL C01640 V=800.0 PL=0
MOVL C01641 V=800.0 PL=0
MOVL C01642 V=800.0 PL=0
MOVL C01643 V=800.0 PL=0
MOVL C01644 V=800.0 PL=0
MOVL C01645 V=800.0 PL=0
MOVL C01646 V=800.0 PL=0
MOVL C01647 V=800.0 PL=0
MOVL C01648 V=800.0 PL=0
MOVL C01649 V=800.0 PL=0
MOVL C01650 V=800.0 PL=0
MOVL C01651 V=800.0 PL=0
MOVL C01652 V=800.0 PL=0
MOVL C01653 V=800.0 PL=0
MOVL C01654 V=800.0 PL=0
MOVL C01655 V=800.0 PL=0
MOVL C01656 V=800.0 PL=0
MOVL C01657 V=800.0 PL=0
MOVL C01658 V=800.0 PL=0
MOVL C01659 V=800.0 PL=0
MOVL C01660 V=800.0 PL=0
MOVL C01661 V=800.0 PL=0
MOVL C01662 V=800.0 PL=0
MOVL C01663 V=800.0 PL=0
MOVL C01664 V=800.0 PL=0
MOVL C01665 V=800.0 PL=0
MOVL C01666 V=800.0 PL=0
MOVL C01667 V=800.0 PL=0
MOVL C01668 V=800.0 PL=0
MOVL C01669 V=800.0 PL=0
MOVL C01670 V=800.0 PL=0
MOVL C01671 V=800.0 PL=0
MOVL C01672 V=800.0 PL=0
MOVL C01673 V=800.0 PL=0
MOVL C01674 V=800.0 PL=0
MOVL C01675 V=800.0 PL=0
MOVL C01676 V=800.0 PL=0
MOVL C01677 V=800.0 PL=0
MOVL C01678 V=800.0 PL=0
MOVL C01679 V=800.0 PL=0
MOVL C01680 V=800.0 PL=0
MOVL C01681 V=800.0 PL=0
MOVL C01682 V=800.0 PL=0
MOVL C01683 V=800.0 PL=0
MOVL C01684 V=800.0 PL=0
MOVL C01685 V=800.0 PL=0
MOVL C01686 V=800.0 PL=0
MOVL C01687 V=800.0 PL=0
MOVL C01688 V=800.0 PL=0
MOVL C01689 V=800.0 PL=0
MOVL C01690 V=800.0 PL=0
MOVL C01691 V=800.0 PL=0
MOVL C01692 V=800.0 PL=0
MOVL C01693 V=800.0 PL=0
MOVL C01694 V=800.0 PL=0
MOVL C01695 V=800.0 PL=0
MOVL C01696 V=800.0 PL=0
MOVL C01697 V=800.0 PL=0
MOVL C01698 V=800.0 PL=0
MOVL C01699 V=800.0 PL=0
MOVL C01700 V=800.0 PL=0
MOVL C01701 V=800.0 PL=0
MOVL C01702 V=800.0 PL=0
MOVL C01703 V=800.0 PL=0
MOVL C01704 V=800.0 PL=0
MOVL C01705 V=800.0 PL=0
MOVL C01706 V=800.0 PL=0
MOVL C01707 V=800.0 PL=0
MOVL C01708 V=800.0 PL=0
MOVL C01709 V=800.0 PL=0
MOVL C01710 V=800.0 PL=0
MOVL C01711 V=800.0 PL=0
MOVL C01712 V=800.0 PL=0
MOVL C01713 V=800.0 PL=0
MOVL C01714 V=800.0 PL=0
MOVL C01715 V=800.0 PL=0
MOVL C01716 V=800.0 PL=0
MOVL C01717 V=800.0 PL=0
MOVL C01718 V=800.0 PL=0
MOVL C01719 V=800.0 PL=0
MOVL C01720 V=800.0 PL=0
MOVL C01721 V=800.0 PL=0
MOVL C01722 V=800.0 PL=0
MOVL C01723 V=800.0 PL=0
MOVL C01724 V=800.0 PL=0
MOVL C01725 V=800.0 PL=0
MOVL C01726 V=800.0 PL=0
MOVL C01727 V=800.0 PL=0
MOVL C01728 V=800.0 PL=0
MOVL C01729 V=800.0 PL=0
MOVL C01730 V=800.0 PL=0
MOVL C01731 V=800.0 PL=0
MOVL C01732 V=800.0 PL=0
MOVL C01733 V=800.0 PL=0
MOVL C01734 V=800.0 PL=0
MOVL C01735 V=800.0 PL=0
MOVL C01736 V=800.0 PL=0
MOVL C01737 V=800.0 PL=0
MOVL C01738 V=800.0 PL=0
MOVL C01739 V=800.0 PL=0
MOVL C01740 V=800.0 PL=0
MOVL C01741 V=800.0 PL=0
MOVL C01742 V=800.0 PL=0
MOVL C01743 V=800.0 PL=0
MOVL C01744 V=800.0 PL=0
MOVL C01745 V=800.0 PL=0
MOVL C01746 V=800.0 PL=0
MOVL C01747 V=800.0 PL=0
MOVL C01748 V=800.0 PL=0
MOVL C01749 V=800.0 PL=0
MOVL C01750 V=800.0 PL=0
MOVL C01751 V=800.0 PL=0
MOVL C01752 V=800.0 PL=0
MOVL C01753 V=800.0 PL=0
MOVL C01754 V=800.0 PL=0
MOVL C01755 V=800.0 PL=0
MOVL C01756 V=800.0 PL=0
MOVL C01757 V=800.0 PL=0
MOVL C01758 V=800.0 PL=0
MOVL C01759 V=800.0 PL=0
MOVL C01760 V=800.0 PL=0
MOVL C01761 V=800.0 PL=0
MOVL C01762 V=800.0 PL=0
MOVL C01763 V=800.0 PL=0
MOVL C01764 V=800.0 PL=0
MOVL C01765 V=800.0 PL=0
MOVL C01766 V=800.0 PL=0
MOVL C01767 V=800.0 PL=0
MOVL C01768 V=800.0 PL=0
MOVL C01769 V=800.0 PL=0
MOVL C01770 V=800.0 PL=0
MOVL C01771 V=800.0 PL=0
MOVL C01772 V=800.0 PL=0
MOVL C01773 V=800.0 PL=0
MOVL C01774 V=800.0 PL=0
MOVL C01775 V=800.0 PL=0
MOVL C01776 V=800.0 PL=0
MOVL C01777 V=800.0 PL=0
MOVL C01778 V=800.0 PL=0
MOVL C01779 V=800.0 PL=0
MOVL C01780 V=800.0 PL=0
MOVL C01781 V=800.0 PL=0
MOVL C01782 V=800.0 PL=0
MOVL C01783 V=800.0 PL=0
MOVL C01784 V=800.0 PL=0
MOVL C01785 V=800.0 PL=0
MOVL C01786 V=800.0 PL=0
MOVL C01787 V=800.0 PL=0
MOVL C01788 V=800.0 PL=0
MOVL C01789 V=800.0 PL=0
MOVL C01790 V=800.0 PL=0
MOVL C01791 V=800.0 PL=0
MOVL C01792 V=800.0 PL=0
MOVL C01793 V=800.0 PL=0
MOVL C01794 V=800.0 PL=0
MOVL C01795 V=800.0 PL=0
MOVL C01796 V=800.0 PL=0
MOVL C01797 V=800.0 PL=0
MOVL C01798 V=800.0 PL=0
MOVL C01799 V=800.0 PL=0
MOVL C01800 V=800.0 PL=0
MOVL C01801 V=800.0 PL=0
MOVL C01802 V=800.0 PL=0
MOVL C01803 V=800.0 PL=0
MOVL C01804 V=800.0 PL=0
MOVL C01805 V=800.0 PL=0
MOVL C01806 V=800.0 PL=0
MOVL C01807 V=800.0 PL=0
MOVL C01808 V=800.0 PL=0
MOVL C01809 V=800.0 PL=0
MOVL C01810 V=800.0 PL=0
MOVL C01811 V=800.0 PL=0
MOVL C01812 V=800.0 PL=0
MOVL C01813 V=800.0 PL=0
MOVL C01814 V=800.0 PL=0
MOVL C01815 V=800.0 PL=0
MOVL C01816 V=800.0 PL=0
MOVL C01817 V=800.0 PL=0
MOVL C01818 V=800.0 PL=0
MOVL C01819 V=800.0 PL=0
MOVL C01820 V=800.0 PL=0
MOVL C01821 V=800.0 PL=0
MOVL C01822 V=800.0 PL=0
MOVL C01823 V=800.0 PL=0
MOVL C01824 V=800.0 PL=0
MOVL C01825 V=800.0 PL=0
MOVL C01826 V=800.0 PL=0
MOVL C01827 V=800.0 PL=0
MOVL C01828 V=800.0 PL=0
MOVL C01829 V=800.0 PL=0
MOVL C01830 V=800.0 PL=0
MOVL C01831 V=800.0 PL=0
MOVL C01832 V=800.0 PL=0
MOVL C01833 V=800.0 PL=0
MOVL C01834 V=800.0 PL=0
MOVL C01835 V=800.0 PL=0
MOVL C01836 V=800.0 PL=0
MOVL C01837 V=800.0 PL=0
MOVL C01838 V=800.0 PL=0
MOVL C01839 V=800.0 PL=0
MOVL C01840 V=800.0 PL=0
MOVL C01841 V=800.0 PL=0
MOVL C01842 V=800.0 PL=0
MOVL C01843 V=800.0 PL=0
MOVL C01844 V=800.0 PL=0
MOVL C01845 V=800.0 PL=0
MOVL C01846 V=800.0 PL=0
MOVL C01847 V=800.0 PL=0
MOVL C01848 V=800.0 PL=0
MOVL C01849 V=800.0 PL=0
MOVL C01850 V=800.0 PL=0
MOVL C01851 V=800.0 PL=0
MOVL C01852 V=800.0 PL=0
MOVL C01853 V=800.0 PL=0
MOVL C01854 V=800.0 PL=0
MOVL C01855 V=800.0 PL=0
MOVL C01856 V=800.0 PL=0
MOVL C01857 V=800.0 PL=0
MOVL C01858 V=800.0 PL=0
MOVL C01859 V=800.0 PL=0
MOVL C01860 V=800.0 PL=0
MOVL C01861 V=800.0 PL=0
MOVL C01862 V=800.0 PL=0
MOVL C01863 V=800.0 PL=0
MOVL C01864 V=800.0 PL=0
MOVL C01865 V=800.0 PL=0
MOVL C01866 V=800.0 PL=0
MOVL C01867 V=800.0 PL=0
MOVL C01868 V=800.0 PL=0
MOVL C01869 V=800.0 PL=0
MOVL C01870 V=800.0 PL=0
MOVL C01871 V=800.0 PL=0
MOVL C01872 V=800.0 PL=0
MOVL C01873 V=800.0 PL=0
MOVL C01874 V=800.0 PL=0
MOVL C01875 V=800.0 PL=0
MOVL C01876 V=800.0 PL=0
MOVL C01877 V=800.0 PL=0
MOVL C01878 V=800.0 PL=0
MOVL C01879 V=800.0 PL=0
MOVL C01880 V=800.0 PL=0
MOVL C01881 V=800.0 PL=0
MOVL C01882 V=800.0 PL=0
MOVL C01883 V=800.0 PL=0
MOVL C01884 V=800.0 PL=0
MOVL C01885 V=800.0 PL=0
MOVL C01886 V=800.0 PL=0
MOVL C01887 V=800.0 PL=0
MOVL C01888 V=800.0 PL=0
MOVL C01889 V=800.0 PL=0
MOVL C01890 V=800.0 PL=0
MOVL C01891 V=800.0 PL=0
MOVL C01892 V=800.0 PL=0
MOVL C01893 V=800.0 PL=0
MOVL C01894 V=800.0 PL=0
MOVL C01895 V=800.0 PL=0
MOVL C01896 V=800.0 PL=0
MOVL C01897 V=800.0 PL=0
MOVL C01898 V=800.0 PL=0
MOVL C01899 V=800.0 PL=0
MOVL C01900 V=800.0 PL=0
MOVL C01901 V=800.0 PL=0
MOVL C01902 V=800.0 PL=0
MOVL C01903 V=800.0 PL=0
MOVL C01904 V=800.0 PL=0
MOVL C01905 V=800.0 PL=0
MOVL C01906 V=800.0 PL=0
MOVL C01907 V=800.0 PL=0
MOVL C01908 V=800.0 PL=0
MOVL C01909 V=800.0 PL=0
MOVL C01910 V=800.0 PL=0
MOVL C01911 V=800.0 PL=0
MOVL C01912 V=800.0 PL=0
MOVL C01913 V=800.0 PL=0
MOVL C01914 V=800.0 PL=0
MOVL C01915 V=800.0 PL=0
MOVL C01916 V=800.0 PL=0
MOVL C01917 V=800.0 PL=0
MOVL C01918 V=800.0 PL=0
MOVL C01919 V=800.0 PL=0
MOVL C01920 V=800.0 PL=0
MOVL C01921 V=800.0 PL=0
MOVL C01922 V=800.0 PL=0
MOVL C01923 V=800.0 PL=0
MOVL C01924 V=800.0 PL=0
MOVL C01925 V=800.0 PL=0
MOVL C01926 V=800.0 PL=0
MOVL C01927 V=800.0 PL=0
MOVL C01928 V=800.0 PL=0
MOVL C01929 V=800.0 PL=0
MOVL C01930 V=800.0 PL=0
MOVL C01931 V=800.0 PL=0
MOVL C01932 V=800.0 PL=0
MOVL C01933 V=800.0 PL=0
MOVL C01934 V=800.0 PL=0
MOVL C01935 V=800.0 PL=0
MOVL C01936 V=800.0 PL=0
MOVL C01937 V=800.0 PL=0
MOVL C01938 V=800.0 PL=0
MOVL C01939 V=800.0 PL=0
MOVL C01940 V=800.0 PL=0
MOVL C01941 V=800.0 PL=0
MOVL C01942 V=800.0 PL=0
MOVL C01943 V=800.0 PL=0
MOVL C01944 V=800.0 PL=0
MOVL C01945 V=800.0 PL=0
MOVL C01946 V=800.0 PL=0
MOVL C01947 V=800.0 PL=0
MOVL C01948 V=800.0 PL=0
MOVL C01949 V=800.0 PL=0
MOVL C01950 V=800.0 PL=0
MOVL C01951 V=800.0 PL=0
MOVL C01952 V=800.0 PL=0
MOVL C01953 V=800.0 PL=0
MOVL C01954 V=800.0 PL=0
MOVL C01955 V=800.0 PL=0
MOVL C01956 V=800.0 PL=0
MOVL C01957 V=800.0 PL=0
MOVL C01958 V=800.0 PL=0
MOVL C01959 V=800.0 PL=0
MOVL C01960 V=800.0 PL=0
MOVL C01961 V=800.0 PL=0
MOVL C01962 V=800.0 PL=0
MOVL C01963 V=800.0 PL=0
MOVL C01964 V=800.0 PL=0
MOVL C01965 V=800.0 PL=0
MOVL C01966 V=800.0 PL=0
MOVL C01967 V=800.0 PL=0
MOVL C01968 V=800.0 PL=0
MOVL C01969 V=800.0 PL=0
MOVL C01970 V=800.0 PL=0
MOVL C01971 V=800.0 PL=0
MOVL C01972 V=800.0 PL=0
MOVL C01973 V=800.0 PL=0
MOVL C01974 V=800.0 PL=0
MOVL C01975 V=800.0 PL=0
MOVL C01976 V=800.0 PL=0
MOVL C01977 V=800.0 PL=0
MOVL C01978 V=800.0 PL=0
MOVL C01979 V=800.0 PL=0
MOVL C01980 V=800.0 PL=0
MOVL C01981 V=800.0 PL=0
MOVL C01982 V=800.0 PL=0
MOVL C01983 V=800.0 PL=0
MOVL C01984 V=800.0 PL=0
MOVL C01985 V=800.0 PL=0
MOVL C01986 V=800.0 PL=0
MOVL C01987 V=800.0 PL=0
MOVL C01988 V=800.0 PL=0
MOVL C01989 V=800.0 PL=0
MOVL C01990 V=800.0 PL=0
MOVL C01991 V=800.0 PL=0
MOVL C01992 V=800.0 PL=0
MOVL C01993 V=800.0 PL=0
MOVL C01994 V=800.0 PL=0
MOVL C01995 V=800.0 PL=0
MOVL C01996 V=800.0 PL=0
MOVL C01997 V=800.0 PL=0
MOVL C01998 V=800.0 PL=0
MOVL C01999 V=800.0 PL=0
MOVL C02000 V=800.0 PL=0
MOVL C02001 V=800.0 PL=0
MOVL C02002 V=800.0 PL=0
MOVL C02003 V=800.0 PL=0
MOVL C02004 V=800.0 PL=0
MOVL C02005 V=800.0 PL=0
MOVL C02006 V=800.0 PL=0
MOVL C02007 V=800.0 PL=0
MOVL C02008 V=800.0 PL=0
MOVL C02009 V=800.0 PL=0
MOVL C02010 V=800.0 PL=0
MOVL C02011 V=800.0 PL=0
MOVL C02012 V=800.0 PL=0
MOVL C02013 V=800.0 PL=0
MOVL C02014 V=800.0 PL=0
MOVL C02015 V=800.0 PL=0
MOVL C02016 V=800.0 PL=0
MOVL C02017 V=800.0 PL=0
MOVL C02018 V=800.0 PL=0
MOVL C02019 V=800.0 PL=0
MOVL C02020 V=800.0 PL=0
MOVL C02021 V=800.0 PL=0
MOVL C02022 V=800.0 PL=0
MOVL C02023 V=800.0 PL=0
MOVL C02024 V=800.0 PL=0
MOVL C02025 V=800.0 PL=0
MOVL C02026 V=800.0 PL=0
MOVL C02027 V=800.0 PL=0
MOVL C02028 V=800.0 PL=0
MOVL C02029 V=800.0 PL=0
MOVL C02030 V=800.0 PL=0
MOVL C02031 V=800.0 PL=0
MOVL C02032 V=800.0 PL=0
MOVL C02033 V=800.0 PL=0
MOVL C02034 V=800.0 PL=0
MOVL C02035 V=800.0 PL=0
MOVL C02036 V=800.0 PL=0
MOVL C02037 V=800.0 PL=0
